CODESYSSPV3/3S/IecVarAccess;String;|var|CODESYS Control Win V3 x64.Application.IOs.SOP720_Pal_Full;Read;SOP720_Pal_Full;Digital;;
CODESYSSPV3/3S/IecVarAccess;String;|var|CODESYS Control Win V3 x64.Application.IOs.SOP720_Pal_Refill;Read;SOP720_Pal_Refill;Digital;;
CODESYSSPV3/3S/IecVarAccess;String;|var|CODESYS Control Win V3 x64.Application.IOs.SOP720_Pal_Dispense;Read;SOP720_Pal_Dispense;Digital;;
CODESYSSPV3/3S/IecVarAccess;String;|var|CODESYS Control Win V3 x64.Application.IOs.SOP721_KM1;Read;SOP721_KM1;Digital;;
CODESYSSPV3/3S/IecVarAccess;String;|var|CODESYS Control Win V3 x64.Application.IOs.SOP721_KM2;Read;SOP721_KM2;Digital;;
CODESYSSPV3/3S/IecVarAccess;String;|var|CODESYS Control Win V3 x64.Application.IOs.SOP730_KM1;Read;SOP730_KM1;Digital;;
CODESYSSPV3/3S/IecVarAccess;String;|var|CODESYS Control Win V3 x64.Application.IOs.SOP730_KM2;Read;SOP730_KM2;Digital;;
CODESYSSPV3/3S/IecVarAccess;String;|var|CODESYS Control Win V3 x64.Application.IOs.SOP730_K2;Read;SOP730_K2;Digital;;
CODESYSSPV3/3S/IecVarAccess;String;|var|CODESYS Control Win V3 x64.Application.IOs.SOP730_K3;Read;SOP730_K3;Digital;;
CODESYSSPV3/3S/IecVarAccess;String;|var|CODESYS Control Win V3 x64.Application.IOs.SOP730_K4;Read;SOP730_K4;Digital;;
CODESYSSPV3/3S/IecVarAccess;String;|var|CODESYS Control Win V3 x64.Application.IOs.SOP730_K5;Read;SOP730_K5;Digital;;
CODESYSSPV3/3S/IecVarAccess;String;|var|CODESYS Control Win V3 x64.Application.IOs.SOP722_KM1;Read;SOP722_KM1;Digital;;
CODESYSSPV3/3S/IecVarAccess;String;|var|CODESYS Control Win V3 x64.Application.IOs.SOP722_KM2;Read;SOP722_KM2;Digital;;
CODESYSSPV3/3S/IecVarAccess;String;|var|CODESYS Control Win V3 x64.Application.IOs.SOP723_KM1;Read;SOP723_KM1;Digital;;
CODESYSSPV3/3S/IecVarAccess;String;|var|CODESYS Control Win V3 x64.Application.IOs.SOP723_KM2;Read;SOP723_KM2;Digital;;
CODESYSSPV3/3S/IecVarAccess;String;|var|CODESYS Control Win V3 x64.Application.IOs.SOP723_K1;Read;SOP723_K1;Digital;;
CODESYSSPV3/3S/IecVarAccess;String;|var|CODESYS Control Win V3 x64.Application.IOs.SOP723_K2;Read;SOP723_K2;Digital;;
CODESYSSPV3/3S/IecVarAccess;String;|var|CODESYS Control Win V3 x64.Application.IOs.SOP740_PickProduct;Read;SOP740_PickProduct;Digital;;
CODESYSSPV3/3S/IecVarAccess;String;|var|CODESYS Control Win V3 x64.Application.IOs.SOP750_K3;Read;SOP750_K3;Digital;;
CODESYSSPV3/3S/IecVarAccess;String;|var|CODESYS Control Win V3 x64.Application.IOs.SOP750_K4;Read;SOP750_K4;Digital;;
CODESYSSPV3/3S/IecVarAccess;String;|var|CODESYS Control Win V3 x64.Application.IOs.SOP750_K5;Read;SOP750_K5;Digital;;
CODESYSSPV3/3S/IecVarAccess;String;|var|CODESYS Control Win V3 x64.Application.IOs.SOP750_K6;Read;SOP750_K6;Digital;;
CODESYSSPV3/3S/IecVarAccess;String;|var|CODESYS Control Win V3 x64.Application.IOs.SOP700_Faulted;Read;SOP700_Faulted;Digital;;
CODESYSSPV3/3S/IecVarAccess;String;|var|CODESYS Control Win V3 x64.Application.IOs.SOP740_Pal_Pos_1;Read;SOP740_Pal_Pos_1;Digital;;
CODESYSSPV3/3S/IecVarAccess;String;|var|CODESYS Control Win V3 x64.Application.IOs.SOP740_Pal_Pos_2;Read;SOP740_Pal_Pos_2;Digital;;
CODESYSSPV3/3S/IecVarAccess;String;|var|CODESYS Control Win V3 x64.Application.IOs.SOP740_Pal_Pos_3;Read;SOP740_Pal_Pos_3;Digital;;
CODESYSSPV3/3S/IecVarAccess;String;|var|CODESYS Control Win V3 x64.Application.IOs.SOP700_H1;Read;SOP700_H1;Digital;;
CODESYSSPV3/3S/IecVarAccess;String;|var|CODESYS Control Win V3 x64.Application.IOs.SOP700_H4;Read;SOP700_H4;Digital;;
CODESYSSPV3/3S/IecVarAccess;String;|var|CODESYS Control Win V3 x64.Application.IOs.SOP700_H7;Read;SOP700_H7;Digital;;
CODESYSSPV3/3S/IecVarAccess;String;|var|CODESYS Control Win V3 x64.Application.IOs.SOP700_H10;Read;SOP700_H10;Digital;;
CODESYSSPV3/3S/IecVarAccess;String;|var|CODESYS Control Win V3 x64.Application.IOs.SOP700_H11;Read;SOP700_H11;Digital;;
CODESYSSPV3/3S/IecVarAccess;String;|var|CODESYS Control Win V3 x64.Application.IOs.SOP700_H14;Read;SOP700_H14;Digital;;
CODESYSSPV3/3S/IecVarAccess;String;|var|CODESYS Control Win V3 x64.Application.IOs.SOP700_H15;Read;SOP700_H15;Digital;;
CODESYSSPV3/3S/IecVarAccess;String;|var|CODESYS Control Win V3 x64.Application.IOs.SOP700_H16;Read;SOP700_H16;Digital;;
CODESYSSPV3/3S/IecVarAccess;String;|var|CODESYS Control Win V3 x64.Application.IOs.SOP740_ProductNr;Read;SOP740_ProductNr;Group;;
CODESYSSPV3/3S/IecVarAccess;String;|var|CODESYS Control Win V3 x64.Application.IOs.SOP723_RetirePallet;Read;SOP723_RetirePallet;Digital;;
CODESYSSPV3/3S/IecVarAccess;String;|var|CODESYS Control Win V3 x64.Application.IOs.SOP720_K5;Read;SOP720_K5;Digital;;
CODESYSSPV3/3S/IecVarAccess;String;|var|CODESYS Control Win V3 x64.Application.IOs.SOP720_K6;Read;SOP720_K6;Digital;;
CODESYSSPV3/3S/IecVarAccess;String;|var|CODESYS Control Win V3 x64.Application.IOs.SOP720_DispensorUp;Write;SOP720_DispensorUp;Digital;;
CODESYSSPV3/3S/IecVarAccess;String;|var|CODESYS Control Win V3 x64.Application.IOs.SOP720_DispensorMid;Write;SOP720_DispensorMid;Digital;;
CODESYSSPV3/3S/IecVarAccess;String;|var|CODESYS Control Win V3 x64.Application.IOs.SOP720_DispensorDown;Write;SOP720_DispensorDown;Digital;;
CODESYSSPV3/3S/IecVarAccess;String;|var|CODESYS Control Win V3 x64.Application.IOs.SOP720_Pal_DispenseDown;Read;SOP720_Pal_DispenseDown;Digital;;
CODESYSSPV3/3S/IecVarAccess;String;|var|CODESYS Control Win V3 x64.Application.IOs.Box_ProductNr;Write;Box_ProductNr;Group;;
CODESYSSPV3/3S/IecVarAccess;String;|var|CODESYS Control Win V3 x64.Application.IOs.Box_IDNumber;Write;Box_IDNumber;Group;;
CODESYSSPV3/3S/IecVarAccess;String;|var|CODESYS Control Win V3 x64.Application.IOs.Status;Write;Status;Group;;

  - Light Curtain Sensor 1 [smart component] at (-31.6, 0, -77.53) mm
      signals: DI DisableSensor, DO Detection
      connections:
        PlaneSensor.SensorOut -> Light Curtain Sensor 1.Detection
        Light Curtain Sensor 1.DisableSensor -> Hide.Execute
        Light Curtain Sensor 1.DisableSensor -> LogicGate_3.InputA
        LogicGate_3.Output -> Show.Execute
        Light Curtain Sensor 1.DisableSensor -> LogicGate_4.InputA
        LogicGate_4.Output -> PlaneSensor.Active
    - PlaneSensor [smart component, from Components\PlaneSensor.rslib] at (2884.52, 14026.71, 333.51) mm, rotated rx 180 ry 0 rz 0 deg
        properties: Origin=[2.28654003266257 4.4307927432671 0.0338898089966275]; Axis1=[2.3 0 0]; Axis2=[0 0 -1.4]; Tag=(none); SensedPart=(none)
      - _sensorPart_ [part], size 2300 x 0 x 1400 mm
    - Show [smart component, from Components\Show.rslib]
        properties: Object=PlaneSensor
    - Hide [smart component, from Components\Hide.rslib]
        properties: Object=PlaneSensor
    - LogicGate_3 [smart component, from Components\LogicGate.rslib]
        properties: Operator=NOT; Delay=0
    - LogicGate_4 [smart component, from Components\LogicGate.rslib]
        properties: Operator=NOT; Delay=0
  - Light Curtain Sensor 2 [smart component] at (0, -1819.31, 0) mm
      signals: DI DisableSensor, DO Detection
      connections:
        PlaneSensor_2.SensorOut -> Light Curtain Sensor 2.Detection
        Light Curtain Sensor 2.DisableSensor -> Show_2.Execute
        Light Curtain Sensor 2.DisableSensor -> LogicGate_4.InputA
        Light Curtain Sensor 2.DisableSensor -> Hide_2.Execute
        LogicGate_4.Output -> Show.Execute
        Light Curtain Sensor 2.DisableSensor -> LogicGate_5.InputA
        LogicGate_5.Output -> PlaneSensor_2.Active
    - PlaneSensor_2 [smart component, from Components\PlaneSensor.rslib] at (0, 0, 396.73) mm
        properties: Origin=[5.139461 9.59591 0.22208]; Axis1=[2.3 0 0]; Axis2=[0 0 1]; Tag=(none); SensedPart=(none)
      - _sensorPart_ [part], size 2300 x 0 x 1000 mm
    - Hide_2 [smart component, from Components\Hide.rslib]
        properties: Object=PlaneSensor_2
    - LogicGate_4 [smart component, from Components\LogicGate.rslib]
        properties: Operator=NOT; Delay=0
    - Show [smart component, from Components\Show.rslib]
        properties: Object=PlaneSensor_2
    - LogicGate_5 [smart component, from Components\LogicGate.rslib]
        properties: Operator=NOT; Delay=0
  - Light Curtain Sensor 3 [smart component] at (0, -6989.64, 0) mm
      signals: DI DisableSensor, DO Detection
      connections:
        PlaneSensor_3.SensorOut -> Light Curtain Sensor 3.Detection
        LogicGate_5.Output -> Show_3.Execute
        Light Curtain Sensor 3.DisableSensor -> Hide_3.Execute
        Light Curtain Sensor 3.DisableSensor -> LogicGate_5.InputA
        LogicGate_5.Output -> PlaneSensor_3.Active
    - PlaneSensor_3 [smart component, from Components\PlaneSensor.rslib] at (-89.72, 0, 389.63) mm
        properties: Origin=[5.139461 9.59591 0.22208]; Axis1=[2.4 0 0]; Axis2=[0 0 1]; Tag=(none); SensedPart=(none)
      - _sensorPart_ [part], size 2400 x 0 x 1000 mm
    - LogicGate_5 [smart component, from Components\LogicGate.rslib]
        properties: Operator=NOT; Delay=0
    - Show_3 [smart component, from Components\Show.rslib]
        properties: Object=PlaneSensor_3
    - Hide_3 [smart component, from Components\Hide.rslib]
        properties: Object=PlaneSensor_3
  - Light Curtain Sensor 4 [smart component] at (17259.69, -4413.54, -135.54) mm, rotated rx 0 ry 0 rz 90 deg
      signals: DI DisableSensor, DO Detection
      connections:
        PlaneSensor_4.SensorOut -> Light Curtain Sensor 4.Detection
        Light Curtain Sensor 4.DisableSensor -> Hide_4.Execute
        Light Curtain Sensor 4.DisableSensor -> LogicGate_6.InputA
        LogicGate_6.Output -> Show_4.Execute
        LogicGate_6.Output -> PlaneSensor_4.Active
    - PlaneSensor_4 [smart component, from Components\PlaneSensor.rslib] at (-119.79, 209.38, 385.64) mm
        properties: Origin=[5.139461 9.59591 0.22208]; Axis1=[2 0 0]; Axis2=[0 0 1.15]; Tag=(none); SensedPart=(none)
      - _sensorPart_ [part], size 2000 x 0 x 1150 mm
    - Hide_4 [smart component, from Components\Hide.rslib]
        properties: Object=PlaneSensor_4
    - Show_4 [smart component, from Components\Show.rslib]
        properties: Object=PlaneSensor_4
    - LogicGate_6 [smart component, from Components\LogicGate.rslib]
        properties: Operator=NOT; Delay=0
  - Timer [smart component, from Components\Timer.rslib]
      properties: StartTime=0; Interval=0; Repeat=true; CurrentTime=6.024
  - MB16 [part] at (-390.31, 2938.54, 153.88) mm, rotated rx -90 ry 0 rz -174.01 deg, size 307.8 x 156.9 x 705.9 mm
  - MB20 [part] at (-193.15, 1001.07, 153.01) mm, rotated rx 0 ry -90 rz 87.74 deg, size 307.4 x 156.7 x 856 mm
  - MB24 [part] at (1.3, -34.41, 112.44) mm, rotated rx 102.56 ry 0 rz -2.8 deg, size 308.5 x 176.3 x 856.1 mm
  - MB16T [part] at (28.49, 2049.11, 116.85) mm, rotated rx 90 ry 0 rz 104.11 deg, size 705.9 x 158.8 x 305.9 mm
  - SOP722 [smart component] at (6333.61, 6970, 616.89) mm, rotated rx 0 ry 0 rz 90 deg
      properties: ForwardSpeed=0.05; ReverseSpeed=-0.05; ConveyorSpeed=0; SpeedForward=0.7; Constant=1E-09; SpeedBackward=-0.6
      signals: DI MotorFWD, DI MotorREV, DO ConveyorError, DI ResetError, DO MotorFeedback, DO BoxSensor
      connections:
        SOP722.MotorFWD -> ?.Enabled
        SOP722.MotorREV -> ?.Enabled
        ?.Output -> ?.Enabled
        SOP722.MotorFWD -> ?.Execute
        SOP722.MotorREV -> ?.Execute
        SOP722.MotorFWD -> ?.A
        SOP722.MotorREV -> ?.B
        ?.Result -> ConveyorSurfaceBehaviour.SurfaceVelocity
        ?.Output -> ConveyorSurfaceBehaviour.SurfaceVelocity
        ?.Output -> ?.InputA
        ?.Output -> ?.InputB
        SOP722.MotorFWD -> ?.InputA
        SOP722.MotorFWD -> ?.InputA
        SOP722.MotorREV -> ?.InputB
        SOP722.MotorFWD -> ?.InputA
        SOP722.MotorFWD -> ?.A
        ?.Result -> ConveyorSurfaceBehaviour.SurfaceVelocity
        SOP722.MotorFWD -> ?.Set
        SOP722.MotorREV -> ?.Set
        SetIdleSpeed.Result -> SetIdleSpeedToConveyor.Execute
        SOP722.MotorFWD -> SetIdleSpeed.A
        SOP722.MotorREV -> SetIdleSpeed.B
        SOP722.MotorFWD -> SetMotorSafetyBreaker.FWD
        SOP722.MotorREV -> SetMotorSafetyBreaker.REV
        ErrorCheckAndBlockingMotorsAndErrorResetLogic.Output -> SetIdleSpeedToConveyor.Execute
        SOP722.ResetError -> ErrorCheckAndBlockingMotorsAndErrorResetLogic.Reset
        SOP722.MotorFWD -> NoErrorAllowFWD.FWD
        ErrorCheckAndBlockingMotorsAndErrorResetLogic.Output -> NoErrorAllowFWD.Error
        NoErrorAllowFWD.Result -> SetForwardSpeedToConveyor.Execute
        SOP722.MotorREV -> NoErrorAllowREV.REV
        ErrorCheckAndBlockingMotorsAndErrorResetLogic.Output -> NoErrorAllowREV.Error
        NoErrorAllowREV.Result -> SetBackwardSpeedToConveyor.Execute
        SetMotorSafetyBreaker.Result -> ErrorCheckAndBlockingMotorsAndErrorResetLogic.Set
        GraphicsHideLogic.Result -> GraphicsHide.Execute
        SOP722.MotorFWD -> GraphicsHideLogic.FWD
        SOP722.MotorREV -> GraphicsHideLogic.REV
        SOP722.MotorFWD -> MotorFeedbackSignalLogic.A
        SOP722.MotorREV -> MotorFeedbackSignalLogic.A
        ErrorCheckAndBlockingMotorsAndErrorResetLogic.Output -> MotorFeedbackSignalLogic.B
        MotorFeedbackSignalLogic.Result -> SOP722.MotorFeedback
        MotorFeedbackSignalLogic.Result -> GraphicsShow.Execute
        ErrorCheckAndBlockingMotorsAndErrorResetLogic.InvOutput -> SOP722.ConveyorError
        SUB100_B1.SensorSignal -> SOP722.BoxSensor
        ?.Result => ?.Count
        ?.Value => ConveyorSurfaceBehaviour.SurfaceVelocity
        ?.Value => ConveyorSurfaceBehaviour.SurfaceVelocity
        ?.Value => ConveyorSurfaceBehaviour.SurfaceVelocity
        ?.Value => ConveyorSurfaceBehaviour.SurfaceVelocity
        ?.Value => ConveyorSurfaceBehaviour.SurfaceVelocity
        ?.Value => ConveyorSurfaceBehaviour.SurfaceVelocity
        SetIdleSpeedToConveyor.Value => ConveyorSurfaceBehaviour.SurfaceVelocity
        SetForwardSpeedToConveyor.Value => ConveyorSurfaceBehaviour.SurfaceVelocity
        SetBackwardSpeedToConveyor.Value => ConveyorSurfaceBehaviour.SurfaceVelocity
        ?.Result => SetForwardSpeedToConveyor.Max
        ?.A => SetBackwardSpeedToConveyor.Min
        ?.Result => SetBackwardSpeedToConveyor.Max
        ?.A => SetForwardSpeedToConveyor.Min
        GraphicsShow.Object => GraphicsHide.Object
        ?.Object => ?.Object
    - ConveyorSurfaceBehaviour [smart component, from Components\PhysicsControl.rslib] at (-850.96, -505.17, -100) mm
        properties: Object=ConveyorSurface; Behavior=2; SurfaceVelocity=0.500000000078149
    - SetIdleSpeedToConveyor [smart component, from Components\Random.rslib] at (-850.96, -505.17, -100) mm
        properties: Value=3.63538950385311E-14; Min=0; Max=1E-13
    - SetBackwardSpeedToConveyor [smart component, from Components\Random.rslib] at (-850.96, -505.17, -100) mm
        properties: Value=-0.699999999999963; Min=-0.7; Max=-0.6999999999999
    - SetForwardSpeedToConveyor [smart component, from Components\Random.rslib] at (-850.96, -505.17, -100) mm
        properties: Value=0.500000000078149; Min=0.5; Max=0.5000000001
    - SetIdleSpeed [smart component, from Components\LogicExpression.rslib] at (-850.96, -505.17, -100) mm
        properties: Expression=not A and not B
    - SetMotorSafetyBreaker [smart component, from Components\LogicExpression.rslib] at (-850.96, -505.17, -100) mm
        properties: Expression=FWD and REV
    - ErrorCheckAndBlockingMotorsAndErrorResetLogic [smart component, from Components\LogicSRLatch.rslib] at (-850.96, -505.17, -100) mm
    - NoErrorAllowFWD [smart component, from Components\LogicExpression.rslib] at (-850.96, -505.17, -100) mm
        properties: Expression=FWD and not Error
    - NoErrorAllowREV [smart component, from Components\LogicExpression.rslib] at (-850.96, -505.17, -100) mm
        properties: Expression=REV and not Error
    - GraphicsShow [smart component, from Components\Show.rslib] at (-850.96, -505.17, -100) mm
        properties: Object=OnOffGfx
    - GraphicsHide [smart component, from Components\Hide.rslib] at (-850.96, -505.17, -100) mm
        properties: Object=OnOffGfx
    - GraphicsHideLogic [smart component, from Components\LogicExpression.rslib] at (-850.96, -505.17, -100) mm
        properties: Expression=not FWD and not REV
    - GraphicsObjects [graphiccomponentgroup] at (-65.23, -0.94, 0) mm, rotated rx 0 ry 0 rz -90 deg
      - OnOffGfx [graphiccomponentgroup] at (514.42, -850.96, -110.92) mm, rotated rx 0 ry 0 rz 90 deg
        - Part_5 [part] at (-19.01, -85.34, -416.89) mm, rotated rx 0 ry 0 rz -90 deg, size 50 x 1701.5 x 100 mm
        - Part_6 [part] at (0, 1062.79, 0) mm, rotated rx 0 ry 0 rz -90 deg, size 50 x 1701.5 x 100 mm
      - ConveyorSurface [part] at (505.17, -850.96, -112.36) mm, rotated rx 0 ry 0 rz 90 deg, size 1712.3 x 1089.6 x 114.1 mm
    - MotorFeedbackSignalLogic [smart component, from Components\LogicExpression.rslib] at (-850.96, -505.17, -100) mm
        properties: Expression=A AND NOT B
    - Conveyor [part] at (-916.73, -600.7, -162.63) mm, rotated rx 0 ry 0 rz 180 deg, size 1700 x 1300 x 500 mm
    - SUB100_B1 [smart component] at (565.82, 599.25, -101.36) mm, rotated rx 0 ry 0 rz 180 deg
        signals: DO SensorSignal
        connections:
          SensorRay.SensorOut -> ?.Active
          ?.Output -> SUB100_B1.SensorSignal
          SensorRay.SensorOut -> LogicGate.InputA
          GraphicSwitch_2.Output -> LogicGate_2.InputA
          LogicGate_2.Output -> LogicGate.InputB
          LogicGate.Output -> SUB100_B1.SensorSignal
      - SensorRay [smart component, from Components\LineSensor.rslib] at (24.04, 61.94, 174.13) mm
          properties: Start=[0 0 0]; End=[5.26116255894493E-07 0.938058416436489 2.90984203399347E-08]; Radius=0.01; SensedPart=(none); SensedPoint=[0 0 0]; Length=0.938058416436637; Tag=(none)
        - _sensorPart_ [part], size 20 x 938.1 x 20 mm
      - SensorMountWorking [part] at (0, 0, 0) mm, size 50 x 50 x 200 mm
      - GraphicSwitch_2 [smart component, from Components\GraphicSwitch.rslib] at (50, 0, 0) mm
          properties: PartHigh=SensorMountBroken; PartLow=SensorMountWorking
      - SensorMountBroken [part] at (0, 0, 0) mm, size 50 x 50 x 200 mm
      - LogicGate [smart component, from Components\LogicGate.rslib]
          properties: Operator=AND; Delay=0
      - LogicGate_2 [smart component, from Components\LogicGate.rslib]
          properties: Operator=NOT; Delay=0
  - SOP723 [smart component] at (6335.13, 8670, 616.89) mm, rotated rx 0 ry 0 rz 90 deg
      properties: ForwardSpeed=0.05; ReverseSpeed=-0.05; ConveyorSpeed=0; SpeedForward=0.7; Constant=1E-09; SpeedBackward=-0.6
      signals: DI MotorFWD, DI MotorREV, DO ConveyorError, DI ResetError, DO MotorFeedback, DO BoxSensor
      connections:
        SOP723.MotorFWD -> ?.Enabled
        SOP723.MotorREV -> ?.Enabled
        ?.Output -> ?.Enabled
        SOP723.MotorFWD -> ?.Execute
        SOP723.MotorREV -> ?.Execute
        SOP723.MotorFWD -> ?.A
        SOP723.MotorREV -> ?.B
        ?.Result -> ConveyorSurfaceBehaviour.SurfaceVelocity
        ?.Output -> ConveyorSurfaceBehaviour.SurfaceVelocity
        ?.Output -> ?.InputA
        ?.Output -> ?.InputB
        SOP723.MotorFWD -> ?.InputA
        SOP723.MotorFWD -> ?.InputA
        SOP723.MotorREV -> ?.InputB
        SOP723.MotorFWD -> ?.InputA
        SOP723.MotorFWD -> ?.A
        ?.Result -> ConveyorSurfaceBehaviour.SurfaceVelocity
        SOP723.MotorFWD -> ?.Set
        SOP723.MotorREV -> ?.Set
        SetIdleSpeed.Result -> SetIdleSpeedToConveyor.Execute
        SOP723.MotorFWD -> SetIdleSpeed.A
        SOP723.MotorREV -> SetIdleSpeed.B
        SOP723.MotorFWD -> SetMotorSafetyBreaker.FWD
        SOP723.MotorREV -> SetMotorSafetyBreaker.REV
        ErrorCheckAndBlockingMotorsAndErrorResetLogic.Output -> SetIdleSpeedToConveyor.Execute
        SOP723.ResetError -> ErrorCheckAndBlockingMotorsAndErrorResetLogic.Reset
        SOP723.MotorFWD -> NoErrorAllowFWD.FWD
        ErrorCheckAndBlockingMotorsAndErrorResetLogic.Output -> NoErrorAllowFWD.Error
        NoErrorAllowFWD.Result -> SetForwardSpeedToConveyor.Execute
        SOP723.MotorREV -> NoErrorAllowREV.REV
        ErrorCheckAndBlockingMotorsAndErrorResetLogic.Output -> NoErrorAllowREV.Error
        NoErrorAllowREV.Result -> SetBackwardSpeedToConveyor.Execute
        SetMotorSafetyBreaker.Result -> ErrorCheckAndBlockingMotorsAndErrorResetLogic.Set
        GraphicsHideLogic.Result -> GraphicsHide.Execute
        SOP723.MotorFWD -> GraphicsHideLogic.FWD
        SOP723.MotorREV -> GraphicsHideLogic.REV
        SOP723.MotorFWD -> MotorFeedbackSignalLogic.A
        SOP723.MotorREV -> MotorFeedbackSignalLogic.A
        ErrorCheckAndBlockingMotorsAndErrorResetLogic.Output -> MotorFeedbackSignalLogic.B
        MotorFeedbackSignalLogic.Result -> SOP723.MotorFeedback
        MotorFeedbackSignalLogic.Result -> GraphicsShow.Execute
        ErrorCheckAndBlockingMotorsAndErrorResetLogic.InvOutput -> SOP723.ConveyorError
        SUB100_B1.SensorSignal -> SOP723.BoxSensor
        ?.Result => ?.Count
        ?.Value => ConveyorSurfaceBehaviour.SurfaceVelocity
        ?.Value => ConveyorSurfaceBehaviour.SurfaceVelocity
        ?.Value => ConveyorSurfaceBehaviour.SurfaceVelocity
        ?.Value => ConveyorSurfaceBehaviour.SurfaceVelocity
        ?.Value => ConveyorSurfaceBehaviour.SurfaceVelocity
        ?.Value => ConveyorSurfaceBehaviour.SurfaceVelocity
        SetIdleSpeedToConveyor.Value => ConveyorSurfaceBehaviour.SurfaceVelocity
        SetForwardSpeedToConveyor.Value => ConveyorSurfaceBehaviour.SurfaceVelocity
        SetBackwardSpeedToConveyor.Value => ConveyorSurfaceBehaviour.SurfaceVelocity
        ?.Result => SetForwardSpeedToConveyor.Max
        ?.A => SetBackwardSpeedToConveyor.Min
        ?.Result => SetBackwardSpeedToConveyor.Max
        ?.A => SetForwardSpeedToConveyor.Min
        GraphicsShow.Object => GraphicsHide.Object
        ?.Object => ?.Object
    - ConveyorSurfaceBehaviour [smart component, from Components\PhysicsControl.rslib] at (-850.96, -505.17, -100) mm
        properties: Object=ConveyorSurface; Behavior=2; SurfaceVelocity=0.500000000006195
    - SetIdleSpeedToConveyor [smart component, from Components\Random.rslib] at (-850.96, -505.17, -100) mm
        properties: Value=1.83222603138174E-14; Min=0; Max=1E-13
    - SetBackwardSpeedToConveyor [smart component, from Components\Random.rslib] at (-850.96, -505.17, -100) mm
        properties: Value=-0.699999999999983; Min=-0.7; Max=-0.6999999999999
    - SetForwardSpeedToConveyor [smart component, from Components\Random.rslib] at (-850.96, -505.17, -100) mm
        properties: Value=0.500000000006195; Min=0.5; Max=0.5000000001
    - SetIdleSpeed [smart component, from Components\LogicExpression.rslib] at (-850.96, -505.17, -100) mm
        properties: Expression=not A and not B
    - SetMotorSafetyBreaker [smart component, from Components\LogicExpression.rslib] at (-850.96, -505.17, -100) mm
        properties: Expression=FWD and REV
    - ErrorCheckAndBlockingMotorsAndErrorResetLogic [smart component, from Components\LogicSRLatch.rslib] at (-850.96, -505.17, -100) mm
    - NoErrorAllowFWD [smart component, from Components\LogicExpression.rslib] at (-850.96, -505.17, -100) mm
        properties: Expression=FWD and not Error
    - NoErrorAllowREV [smart component, from Components\LogicExpression.rslib] at (-850.96, -505.17, -100) mm
        properties: Expression=REV and not Error
    - GraphicsShow [smart component, from Components\Show.rslib] at (-850.96, -505.17, -100) mm
        properties: Object=OnOffGfx
    - GraphicsHide [smart component, from Components\Hide.rslib] at (-850.96, -505.17, -100) mm
        properties: Object=OnOffGfx
    - GraphicsHideLogic [smart component, from Components\LogicExpression.rslib] at (-850.96, -505.17, -100) mm
        properties: Expression=not FWD and not REV
    - GraphicsObjects [graphiccomponentgroup] at (-65.23, -0.94, 0) mm, rotated rx 0 ry 0 rz -90 deg
      - OnOffGfx [graphiccomponentgroup] at (514.42, -850.96, -110.92) mm, rotated rx 0 ry 0 rz 90 deg
        - Part_5 [part] at (-19.01, -85.34, -416.89) mm, rotated rx 0 ry 0 rz -90 deg, size 50 x 1701.5 x 100 mm
        - Part_6 [part] at (0, 1062.79, 0) mm, rotated rx 0 ry 0 rz -90 deg, size 50 x 1701.5 x 100 mm
      - ConveyorSurface [part] at (505.17, -850.96, -112.36) mm, rotated rx 0 ry 0 rz 90 deg, size 1712.3 x 1089.6 x 114.1 mm
    - MotorFeedbackSignalLogic [smart component, from Components\LogicExpression.rslib] at (-850.96, -505.17, -100) mm
        properties: Expression=A AND NOT B
    - Conveyor [part] at (-916.73, -600.7, -162.63) mm, rotated rx 0 ry 0 rz 180 deg, size 1700 x 1300 x 500 mm
    - SUB100_B1 [smart component] at (565.82, 599.25, -101.36) mm, rotated rx 0 ry 0 rz 180 deg
        signals: DO SensorSignal
        connections:
          SensorRay.SensorOut -> ?.Active
          ?.Output -> SUB100_B1.SensorSignal
          SensorRay.SensorOut -> LogicGate.InputA
          GraphicSwitch_2.Output -> LogicGate_2.InputA
          LogicGate_2.Output -> LogicGate.InputB
          LogicGate.Output -> SUB100_B1.SensorSignal
      - SensorRay [smart component, from Components\LineSensor.rslib] at (24.04, 61.94, 174.13) mm
          properties: Start=[0 0 0]; End=[5.26116255894493E-07 0.938058416436489 2.90984203399347E-08]; Radius=0.01; SensedPart=(none); SensedPoint=[0 0 0]; Length=0.938058416436637; Tag=(none)
        - _sensorPart_ [part], size 20 x 938.1 x 20 mm
      - SensorMountWorking [part] at (0, 0, 0) mm, size 50 x 50 x 200 mm
      - GraphicSwitch_2 [smart component, from Components\GraphicSwitch.rslib] at (50, 0, 0) mm
          properties: PartHigh=SensorMountBroken; PartLow=SensorMountWorking
      - SensorMountBroken [part] at (0, 0, 0) mm, size 50 x 50 x 200 mm
      - LogicGate [smart component, from Components\LogicGate.rslib]
          properties: Operator=AND; Delay=0
      - LogicGate_2 [smart component, from Components\LogicGate.rslib]
          properties: Operator=NOT; Delay=0
  - PalletDispensorMovement [smart component]
      signals: DI ReFillPallet, DI Pallet_FilledUp, DI NewPallet, DO DispensorDown, DO DispensorMid, DO DispensorUp, DI Dispensor_Down, DO DispensorTop
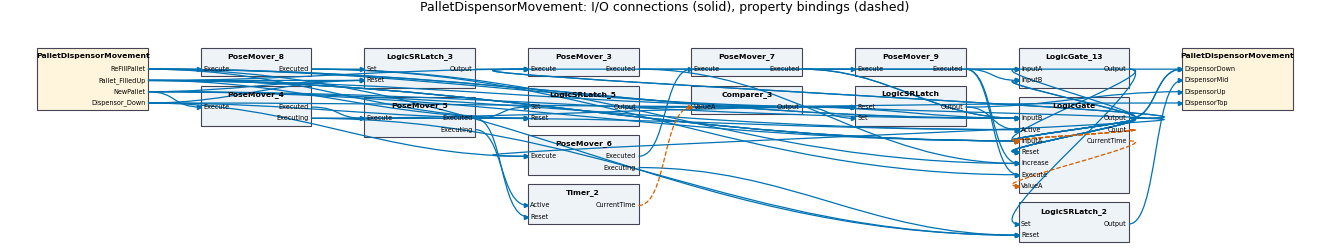
      connections:
        PoseMover_4.Executed -> PoseMover_5.Execute
        PoseMover_6.Executed -> PoseMover_7.Execute
        LogicGate.Output -> PoseMover_3.Execute
        PoseMover_7.Executed -> LogicGate.InputB
        PoseMover_7.Executed -> LogicGate_2.InputB
        LogicGate_2.Output -> PoseMover_3.Execute
        PoseMover_5.Executed -> Timer.Active
        Timer.Output -> PoseMover_6.Execute
        Timer_2.Output -> LogicGate.InputA
        LogicGate.Output -> Timer.Reset
        PalletDispensorMovement.ReFillPallet -> PoseMover_8.Execute
        PalletDispensorMovement.Pallet_FilledUp -> ?.InputA
        PalletDispensorMovement.Pallet_FilledUp -> ?.InputA
        PalletDispensorMovement.Pallet_FilledUp -> PoseMover_3.Execute
        PalletDispensorMovement.NewPallet -> PoseMover_4.Execute
        PalletDispensorMovement.NewPallet -> Timer_2.Active
        PoseMover_7.Executed -> PoseMover_9.Execute
        PoseMover_8.Executed -> Counter_2.Increase
        LogicGate_7.Output -> LogicGate_8.InputA
        LogicGate_8.Output -> Counter_2.Reset
        LogicGate_7.Output -> PalletDispensorMovement.DispensorDown
        PoseMover_9.Executed -> Counter_4.Increase
        LogicGate_11.Output -> LogicGate_12.InputA
        LogicGate_12.Output -> Counter_4.Reset
        PoseMover_3.Executed -> Counter_3.Increase
        LogicGate_9.Output -> LogicGate_10.InputA
        LogicGate_10.Output -> Counter_3.Reset
        LogicGate_9.Output -> LogicGate_13.InputA
        LogicGate_11.Output -> LogicGate_13.InputB
        PoseMover_5.Executing -> Timer_2.Active
        PoseMover_5.Executed -> Timer_2.Reset
        PoseMover_9.Executed -> Repeater.Execute
        Repeater.Output -> LogicGate_13.InputB
        PoseMover_8.Executed -> Repeater_2.Execute
        Repeater_2.Output -> PalletDispensorMovement.DispensorDown
        LogicSRLatch.Output -> Timer_4.Active
        Comparer_4.Output -> LogicSRLatch.Reset
        Comparer_4.Output -> Timer_4.Reset
        LogicSRLatch_3.Output -> PalletDispensorMovement.DispensorDown
        LogicSRLatch_2.Output -> PalletDispensorMovement.DispensorMid
        LogicSRLatch.Output -> PalletDispensorMovement.DispensorUp
        Comparer_3.Output -> LogicSRLatch.Set
        PoseMover_8.Executed -> LogicSRLatch_3.Set
        PoseMover_3.Executed -> LogicGate_13.InputA
        PoseMover_9.Executed -> LogicGate_13.InputB
        LogicGate_13.Output -> LogicSRLatch_2.Set
        LogicGate_13.Output -> LogicGate_15.InputA
        PalletDispensorMovement.ReFillPallet -> LogicGate_15.InputB
        PalletDispensorMovement.Pallet_FilledUp -> LogicGate_14.InputA
        PalletDispensorMovement.NewPallet -> LogicGate_14.InputB
        PalletDispensorMovement.NewPallet -> LogicGate_16.InputA
        PalletDispensorMovement.ReFillPallet -> LogicGate_16.InputB
        LogicGate_16.Output -> LogicGate_17.InputA
        Comparer_3.Output -> LogicGate_17.InputB
        PalletDispensorMovement.Dispensor_Down -> PoseMover_6.Execute
        PoseMover_5.Executed -> LogicSRLatch_5.Set
        LogicSRLatch_5.Output -> PalletDispensorMovement.DispensorTop
        PalletDispensorMovement.ReFillPallet -> LogicSRLatch.Reset
        PalletDispensorMovement.Pallet_FilledUp -> LogicSRLatch.Reset
        PalletDispensorMovement.Dispensor_Down -> LogicSRLatch.Reset
        PoseMover_4.Executing -> LogicSRLatch.Reset
        PalletDispensorMovement.ReFillPallet -> LogicSRLatch_5.Reset
        PalletDispensorMovement.Pallet_FilledUp -> LogicSRLatch_5.Reset
        PalletDispensorMovement.Dispensor_Down -> LogicSRLatch_5.Reset
        PoseMover_4.Executing -> LogicSRLatch_5.Reset
        PalletDispensorMovement.ReFillPallet -> LogicSRLatch_2.Reset
        PoseMover_4.Executing -> LogicSRLatch_2.Reset
        PoseMover_6.Executing -> LogicSRLatch_2.Reset
        PalletDispensorMovement.Pallet_FilledUp -> LogicSRLatch_3.Reset
        PalletDispensorMovement.NewPallet -> LogicSRLatch_3.Reset
        PalletDispensorMovement.Dispensor_Down -> LogicSRLatch_3.Reset
        LogicSRLatch_5.Output -> LogicSRLatch.Reset
        Counter_2.Count => LogicGate_7.InputA
        Counter_4.Count => LogicGate_11.InputA
        Counter_3.Count => LogicGate_9.InputA
        Timer_2.CurrentTime => Comparer_3.ValueA
        Timer_4.CurrentTime => Comparer_4.ValueA
    - PoseMover_3 [smart component, from Components\PoseMover.rslib]
        properties: Mechanism=PalletDispenser; Pose=2; Duration=2
    - PoseMover_4 [smart component, from Components\PoseMover.rslib]
        properties: Mechanism=PalletDispenser; Pose=3; Duration=2
    - PoseMover_5 [smart component, from Components\PoseMover.rslib]
        properties: Mechanism=PalletDispenser; Pose=4; Duration=4
    - PoseMover_6 [smart component, from Components\PoseMover.rslib]
        properties: Mechanism=PalletDispenser; Pose=5; Duration=4
    - PoseMover_7 [smart component, from Components\PoseMover.rslib]
        properties: Mechanism=PalletDispenser; Pose=6; Duration=2
    - PoseMover_8 [smart component, from Components\PoseMover.rslib]
        properties: Mechanism=PalletDispenser; Pose=1; Duration=1
    - PoseMover_9 [smart component, from Components\PoseMover.rslib]
        properties: Mechanism=PalletDispenser; Pose=2; Duration=2
    - LogicGate_13 [smart component, from Components\LogicGate.rslib]
        properties: Operator=OR; Delay=0
    - Timer_2 [smart component, from Components\Timer.rslib]
        properties: StartTime=0; Interval=0; Repeat=true; CurrentTime=0
    - Comparer_3 [smart component, from Components\Comparer.rslib]
        properties: ValueA=0; Operator=>=; ValueB=1
    - LogicSRLatch [smart component, from Components\LogicSRLatch.rslib]
    - LogicSRLatch_2 [smart component, from Components\LogicSRLatch.rslib]
    - LogicSRLatch_3 [smart component, from Components\LogicSRLatch.rslib]
    - LogicSRLatch_5 [smart component, from Components\LogicSRLatch.rslib]
  - PalletDispenser [mechanism] at (0, 0, 0) mm; joint values [0.1316, 0, 0] (rad or m)
      links: Wall, HorizontalBar, LeftClamp, RightClamp
  - EuroPallet (1) [part] at (8313.49, 1114.92, 117.23) mm, rotated rx 0 ry 0 rz 89.94 deg, size 1206.6 x 808.8 x 152.5 mm
  - Buttons [graphiccomponentgroup]
    - FilledPallet [part] at (7471.38, 607.83, 1076.55) mm, rotated rx 0 ry 90 rz 0 deg, size 40 x 39.8 x 10 mm
    - Emergency4 [part] at (7471.38, 607.83, 1236.44) mm, rotated rx 0 ry 90 rz 0 deg, size 40 x 39.8 x 10 mm
    - PalletRemove [part] at (7441.66, 9631.65, 1174.65) mm, rotated rx 0 ry 90 rz 90 deg, size 40 x 39.8 x 10 mm
    - Emergency3 [part] at (7441.66, 9631.65, 1280.76) mm, rotated rx 0 ry 90 rz 90 deg, size 40 x 39.8 x 10 mm
    - Emergency1 [part] at (5192.96, 10430.05, 1449.33) mm, rotated rx 0 ry 90 rz -180 deg, size 40 x 39.8 x 10 mm
    - Emergency2 [part] at (5138.96, 10431.72, 1432.3) mm, rotated rx 0 ry 90 rz -180 deg, size 40 x 39.8 x 10 mm
  - SOP730 [smart component] at (6335.96, 5270, 616.89) mm, rotated rx 0 ry 0 rz 90 deg
      properties: ForwardSpeed=0.05; ReverseSpeed=-0.05; ConveyorSpeed=0; SpeedForward=0.7; Constant=1E-09; SpeedBackward=-0.6
      signals: DI MotorFWD, DI MotorREV, DO ConveyorError, DI ResetError, DO MotorFeedback, DI FrontUp, DI FrontDown, DI RearUp, DI RearDown, DO BoxSensor, DO FrontSensor, DO RearSensor, DO FrontDownSensor, DO RareDownSensor
      connections:
        SOP730.MotorFWD -> ?.Enabled
        SOP730.MotorREV -> ?.Enabled
        ?.Output -> ?.Enabled
        SOP730.MotorFWD -> ?.Execute
        SOP730.MotorREV -> ?.Execute
        SOP730.MotorFWD -> ?.A
        SOP730.MotorREV -> ?.B
        ?.Result -> ConveyorSurfaceBehaviour.SurfaceVelocity
        ?.Output -> ConveyorSurfaceBehaviour.SurfaceVelocity
        ?.Output -> ?.InputA
        ?.Output -> ?.InputB
        SOP730.MotorFWD -> ?.InputA
        SOP730.MotorFWD -> ?.InputA
        SOP730.MotorREV -> ?.InputB
        SOP730.MotorFWD -> ?.InputA
        SOP730.MotorFWD -> ?.A
        ?.Result -> ConveyorSurfaceBehaviour.SurfaceVelocity
        SOP730.MotorFWD -> ?.Set
        SOP730.MotorREV -> ?.Set
        SetIdleSpeed.Result -> SetIdleSpeedToConveyor.Execute
        SOP730.MotorFWD -> SetIdleSpeed.A
        SOP730.MotorREV -> SetIdleSpeed.B
        SOP730.MotorFWD -> SetMotorSafetyBreaker.FWD
        SOP730.MotorREV -> SetMotorSafetyBreaker.REV
        ErrorCheckAndBlockingMotorsAndErrorResetLogic.Output -> SetIdleSpeedToConveyor.Execute
        SOP730.ResetError -> ErrorCheckAndBlockingMotorsAndErrorResetLogic.Reset
        SOP730.MotorFWD -> NoErrorAllowFWD.FWD
        ErrorCheckAndBlockingMotorsAndErrorResetLogic.Output -> NoErrorAllowFWD.Error
        NoErrorAllowFWD.Result -> SetForwardSpeedToConveyor.Execute
        SOP730.MotorREV -> NoErrorAllowREV.REV
        ErrorCheckAndBlockingMotorsAndErrorResetLogic.Output -> NoErrorAllowREV.Error
        NoErrorAllowREV.Result -> SetBackwardSpeedToConveyor.Execute
        SetMotorSafetyBreaker.Result -> ErrorCheckAndBlockingMotorsAndErrorResetLogic.Set
        GraphicsHideLogic.Result -> GraphicsHide.Execute
        SOP730.MotorFWD -> GraphicsHideLogic.FWD
        SOP730.MotorREV -> GraphicsHideLogic.REV
        SOP730.MotorFWD -> MotorFeedbackSignalLogic.A
        SOP730.MotorREV -> MotorFeedbackSignalLogic.A
        ErrorCheckAndBlockingMotorsAndErrorResetLogic.Output -> MotorFeedbackSignalLogic.B
        MotorFeedbackSignalLogic.Result -> SOP730.MotorFeedback
        MotorFeedbackSignalLogic.Result -> GraphicsShow.Execute
        ErrorCheckAndBlockingMotorsAndErrorResetLogic.InvOutput -> SOP730.ConveyorError
        SUB100_B1.SensorSignal -> SOP730.BoxSensor
        SUB730 FrontClamp.ClampUpPosition -> SOP730.FrontSensor
        SUB730 RearClamp.ClampUpPosition -> SOP730.RearSensor
        SOP730.FrontUp -> SUB730 FrontClamp.ClampUp
        SOP730.FrontDown -> SUB730 FrontClamp.ClampDown
        SOP730.RearUp -> SUB730 RearClamp.ClampUp
        SOP730.RearDown -> SUB730 RearClamp.ClampDown
        SOP730.FrontUp -> SUB730 FrontClamp.ClampUp
        SOP730.FrontDown -> SUB730 FrontClamp.ClampDown
        SUB730 FrontClamp.ClampUpPosition -> SOP730.FrontSensor
        SOP730.RearUp -> SUB730 RearClamp.ClampUp
        SOP730.RearDown -> SUB730 RearClamp.ClampDown
        SUB730 RearClamp.ClampUpPosition -> SOP730.RearSensor
        SUB730 FrontClamp.ClampDownPosition -> SOP730.FrontDownSensor
        SUB730 RearClamp.ClampDownPosition -> SOP730.RareDownSensor
        SOP730.FrontUp -> SUB730 FrontClamp.ClampUp
        SOP730.FrontDown -> SUB730 FrontClamp.ClampDown
        SUB730 FrontClamp.ClampUpPosition -> SOP730.FrontSensor
        SUB730 FrontClamp.ClampDownPosition -> SOP730.FrontDownSensor
        ?.Result => ?.Count
        ?.Value => ConveyorSurfaceBehaviour.SurfaceVelocity
        ?.Value => ConveyorSurfaceBehaviour.SurfaceVelocity
        ?.Value => ConveyorSurfaceBehaviour.SurfaceVelocity
        ?.Value => ConveyorSurfaceBehaviour.SurfaceVelocity
        ?.Value => ConveyorSurfaceBehaviour.SurfaceVelocity
        ?.Value => ConveyorSurfaceBehaviour.SurfaceVelocity
        SetIdleSpeedToConveyor.Value => ConveyorSurfaceBehaviour.SurfaceVelocity
        SetForwardSpeedToConveyor.Value => ConveyorSurfaceBehaviour.SurfaceVelocity
        SetBackwardSpeedToConveyor.Value => ConveyorSurfaceBehaviour.SurfaceVelocity
        ?.Result => SetForwardSpeedToConveyor.Max
        ?.A => SetBackwardSpeedToConveyor.Min
        ?.Result => SetBackwardSpeedToConveyor.Max
        ?.A => SetForwardSpeedToConveyor.Min
        GraphicsShow.Object => GraphicsHide.Object
        ?.Object => ?.Object
    - ConveyorSurfaceBehaviour [smart component, from Components\PhysicsControl.rslib] at (-850.96, -505.17, -100) mm
        properties: Object=ConveyorSurface; Behavior=2; SurfaceVelocity=0.500000000050282
    - SetIdleSpeedToConveyor [smart component, from Components\Random.rslib] at (-850.96, -505.17, -100) mm
        properties: Value=6.11436496307811E-14; Min=0; Max=1E-13
    - SetBackwardSpeedToConveyor [smart component, from Components\Random.rslib] at (-850.96, -505.17, -100) mm
        properties: Value=-0.699999999999912; Min=-0.7; Max=-0.6999999999999
    - SetForwardSpeedToConveyor [smart component, from Components\Random.rslib] at (-850.96, -505.17, -100) mm
        properties: Value=0.500000000050282; Min=0.5; Max=0.5000000001
    - SetIdleSpeed [smart component, from Components\LogicExpression.rslib] at (-850.96, -505.17, -100) mm
        properties: Expression=not A and not B
    - SetMotorSafetyBreaker [smart component, from Components\LogicExpression.rslib] at (-850.96, -505.17, -100) mm
        properties: Expression=FWD and REV
    - ErrorCheckAndBlockingMotorsAndErrorResetLogic [smart component, from Components\LogicSRLatch.rslib] at (-850.96, -505.17, -100) mm
    - NoErrorAllowFWD [smart component, from Components\LogicExpression.rslib] at (-850.96, -505.17, -100) mm
        properties: Expression=FWD and not Error
    - NoErrorAllowREV [smart component, from Components\LogicExpression.rslib] at (-850.96, -505.17, -100) mm
        properties: Expression=REV and not Error
    - GraphicsShow [smart component, from Components\Show.rslib] at (-850.96, -505.17, -100) mm
        properties: Object=OnOffGfx
    - GraphicsHide [smart component, from Components\Hide.rslib] at (-850.96, -505.17, -100) mm
        properties: Object=OnOffGfx
    - GraphicsHideLogic [smart component, from Components\LogicExpression.rslib] at (-850.96, -505.17, -100) mm
        properties: Expression=not FWD and not REV
    - GraphicsObjects [graphiccomponentgroup] at (-65.23, -0.94, 0) mm, rotated rx 0 ry 0 rz -90 deg
      - OnOffGfx [graphiccomponentgroup] at (514.42, -850.96, -110.92) mm, rotated rx 0 ry 0 rz 90 deg
        - Part_5 [part] at (-19.01, -85.34, -416.89) mm, rotated rx 0 ry 0 rz -90 deg, size 50 x 1701.5 x 100 mm
        - Part_6 [part] at (0, 1062.79, 0) mm, rotated rx 0 ry 0 rz -90 deg, size 50 x 1701.5 x 100 mm
      - ConveyorSurface [part] at (505.17, -850.96, -112.36) mm, rotated rx 0 ry 0 rz 90 deg, size 1712.3 x 1089.6 x 114.1 mm
    - MotorFeedbackSignalLogic [smart component, from Components\LogicExpression.rslib] at (-850.96, -505.17, -100) mm
        properties: Expression=A AND NOT B
    - Conveyor [part] at (-916.73, -600.7, -162.63) mm, rotated rx 0 ry 0 rz 180 deg, size 1700 x 1300 x 500 mm
    - SUB100_B1 [smart component] at (565.82, 599.25, -101.36) mm, rotated rx 0 ry 0 rz 180 deg
        signals: DO SensorSignal
        connections:
          SensorRay.SensorOut -> ?.Active
          ?.Output -> SUB100_B1.SensorSignal
          SensorRay.SensorOut -> LogicGate.InputA
          GraphicSwitch_2.Output -> LogicGate_2.InputA
          LogicGate_2.Output -> LogicGate.InputB
          LogicGate.Output -> SUB100_B1.SensorSignal
      - SensorRay [smart component, from Components\LineSensor.rslib] at (24.04, 61.94, 174.13) mm
          properties: Start=[0 0 0]; End=[5.26116255894493E-07 0.938058416436489 2.90984203399347E-08]; Radius=0.01; SensedPart=(none); SensedPoint=[0 0 0]; Length=0.938058416436637; Tag=(none)
        - _sensorPart_ [part], size 20 x 938.1 x 20 mm
      - SensorMountWorking [part] at (0, 0, 0) mm, size 50 x 50 x 200 mm
      - GraphicSwitch_2 [smart component, from Components\GraphicSwitch.rslib] at (50, 0, 0) mm
          properties: PartHigh=SensorMountBroken; PartLow=SensorMountWorking
      - SensorMountBroken [part] at (0, 0, 0) mm, size 50 x 50 x 200 mm
      - LogicGate [smart component, from Components\LogicGate.rslib]
          properties: Operator=AND; Delay=0
      - LogicGate_2 [smart component, from Components\LogicGate.rslib]
          properties: Operator=NOT; Delay=0
    - SUB730 RearClamp [smart component, from Components\SUB730 RearClamp1.rslib] at (-679.81, -100.54, -122.63) mm, rotated rx 0 ry 0 rz 90 deg
        connections:
          SUB730 RearClamp.ClampUp -> LogicExpression.A
          BottomPosSensor.SensorOut -> LogicExpression.B
          LogicExpression.Result -> LinearMoveUp.Execute
          SUB730 RearClamp.ClampDown -> LogicExpression_2.A
          BottomPosSensor.SensorOut -> LogicExpression_2.B
          LogicExpression_2.Result -> LinearMoveDown.Execute
          LinearMoveUp.Executed -> LogicSRLatch.Set
          LogicSRLatch.Output -> SUB730 RearClamp.ClampUpPosition
          LinearMoveDown.Executed -> ?.Set
          ?.Output -> SUB730 RearClamp.ClampDownPosition
          LinearMoveDown.Executing -> LogicSRLatch.Reset
          LinearMoveUp.Executing -> ?.Reset
          BottomPosSensor.SensorOut -> SUB730 RearClamp.ClampDownPosition
      - Clamp3D [part, from Components\SUB730 RearClamp1.rslib]
      - BottomPosSensor [smart component, from Components\LineSensor.rslib] at (18.37, 10.91, 93.4) mm
          properties: Start=[-5.44677247749092E-09 -9.84894448774476E-08 -0.0999997155196143]; End=[-5.44677247749092E-09 -9.84894448774476E-08 -0.0899997155196144]; Radius=0.02; SensedPart=Clamp3D; SensedPoint=[6.41812744140625 4.57928466796875 0.49426123046875]; Length=0.0099999999999999; Tag=(none)
        - _sensorPart_ [part, from Components\SUB730 RearClamp1.rslib]
      - LinearMoveUp [smart component, from Components\LinearMover2.rslib]
          properties: Object=Clamp3D; Direction=[0 0 0.1]; Distance=0.1; Duration=1; Reference=Global; ReferenceObject=(none)
      - LinearMoveDown [smart component, from Components\LinearMover2.rslib]
          properties: Object=Clamp3D; Direction=[0 0 -0.1]; Distance=0.1; Duration=1; Reference=Global; ReferenceObject=(none)
      - LogicExpression [smart component, from Components\LogicExpression.rslib]
          properties: Expression=A AND B
      - LogicExpression_2 [smart component, from Components\LogicExpression.rslib]
          properties: Expression=A AND NOT B
      - LogicSRLatch [smart component, from Components\LogicSRLatch.rslib]
    - SUB730 FrontClamp [smart component, from Components\SUB730 RearClamp1.rslib] at (571.35, -100.54, -122.63) mm, rotated rx 0 ry 0 rz 90 deg
        connections:
          SUB730 FrontClamp.ClampUp -> LogicExpression.A
          BottomPosSensor.SensorOut -> LogicExpression.B
          LogicExpression.Result -> LinearMoveUp.Execute
          SUB730 FrontClamp.ClampDown -> LogicExpression_2.A
          BottomPosSensor.SensorOut -> LogicExpression_2.B
          LogicExpression_2.Result -> LinearMoveDown.Execute
          LinearMoveUp.Executed -> LogicSRLatch.Set
          LogicSRLatch.Output -> SUB730 FrontClamp.ClampUpPosition
          LinearMoveDown.Executed -> ?.Set
          ?.Output -> SUB730 FrontClamp.ClampDownPosition
          LinearMoveDown.Executing -> LogicSRLatch.Reset
          LinearMoveUp.Executing -> ?.Reset
          BottomPosSensor.SensorOut -> SUB730 FrontClamp.ClampDownPosition
      - Clamp3D [part, from Components\SUB730 RearClamp1.rslib]
      - BottomPosSensor [smart component, from Components\LineSensor.rslib] at (18.37, 10.91, 93.4) mm
          properties: Start=[-5.44677247749092E-09 -9.84894448774476E-08 -0.0999997155196143]; End=[-5.44677247749092E-09 -9.84894448774476E-08 -0.0899997155196144]; Radius=0.02; SensedPart=Clamp3D; SensedPoint=[6.41812744140625 5.83044482421875 0.494260986328125]; Length=0.0099999999999999; Tag=(none)
        - _sensorPart_ [part, from Components\SUB730 RearClamp1.rslib]
      - LinearMoveUp [smart component, from Components\LinearMover2.rslib]
          properties: Object=Clamp3D; Direction=[0 0 0.1]; Distance=0.1; Duration=1; Reference=Global; ReferenceObject=(none)
      - LinearMoveDown [smart component, from Components\LinearMover2.rslib]
          properties: Object=Clamp3D; Direction=[0 0 -0.1]; Distance=0.1; Duration=1; Reference=Global; ReferenceObject=(none)
      - LogicExpression [smart component, from Components\LogicExpression.rslib]
          properties: Expression=A AND B
      - LogicExpression_2 [smart component, from Components\LogicExpression.rslib]
          properties: Expression=A AND NOT B
      - LogicSRLatch [smart component, from Components\LogicSRLatch.rslib]
  - SOP721 [smart component] at (6333.61, 3570, 616.89) mm, rotated rx 0 ry 0 rz 90 deg
      properties: ForwardSpeed=0.05; ReverseSpeed=-0.05; ConveyorSpeed=0; SpeedForward=0.7; Constant=1E-09; SpeedBackward=-0.6
      signals: DI MotorFWD, DI MotorREV, DO ConveyorError, DI ResetError, DO MotorFeedback, DO BoxSensor
      connections:
        SOP721.MotorFWD -> ?.Enabled
        SOP721.MotorREV -> ?.Enabled
        ?.Output -> ?.Enabled
        SOP721.MotorFWD -> ?.Execute
        SOP721.MotorREV -> ?.Execute
        SOP721.MotorFWD -> ?.A
        SOP721.MotorREV -> ?.B
        ?.Result -> ConveyorSurfaceBehaviour.SurfaceVelocity
        ?.Output -> ConveyorSurfaceBehaviour.SurfaceVelocity
        ?.Output -> ?.InputA
        ?.Output -> ?.InputB
        SOP721.MotorFWD -> ?.InputA
        SOP721.MotorFWD -> ?.InputA
        SOP721.MotorREV -> ?.InputB
        SOP721.MotorFWD -> ?.InputA
        SOP721.MotorFWD -> ?.A
        ?.Result -> ConveyorSurfaceBehaviour.SurfaceVelocity
        SOP721.MotorFWD -> ?.Set
        SOP721.MotorREV -> ?.Set
        SetIdleSpeed.Result -> SetIdleSpeedToConveyor.Execute
        SOP721.MotorFWD -> SetIdleSpeed.A
        SOP721.MotorREV -> SetIdleSpeed.B
        SOP721.MotorFWD -> SetMotorSafetyBreaker.FWD
        SOP721.MotorREV -> SetMotorSafetyBreaker.REV
        ErrorCheckAndBlockingMotorsAndErrorResetLogic.Output -> SetIdleSpeedToConveyor.Execute
        SOP721.ResetError -> ErrorCheckAndBlockingMotorsAndErrorResetLogic.Reset
        SOP721.MotorFWD -> NoErrorAllowFWD.FWD
        ErrorCheckAndBlockingMotorsAndErrorResetLogic.Output -> NoErrorAllowFWD.Error
        NoErrorAllowFWD.Result -> SetForwardSpeedToConveyor.Execute
        SOP721.MotorREV -> NoErrorAllowREV.REV
        ErrorCheckAndBlockingMotorsAndErrorResetLogic.Output -> NoErrorAllowREV.Error
        NoErrorAllowREV.Result -> SetBackwardSpeedToConveyor.Execute
        SetMotorSafetyBreaker.Result -> ErrorCheckAndBlockingMotorsAndErrorResetLogic.Set
        GraphicsHideLogic.Result -> GraphicsHide.Execute
        SOP721.MotorFWD -> GraphicsHideLogic.FWD
        SOP721.MotorREV -> GraphicsHideLogic.REV
        SOP721.MotorFWD -> MotorFeedbackSignalLogic.A
        SOP721.MotorREV -> MotorFeedbackSignalLogic.A
        ErrorCheckAndBlockingMotorsAndErrorResetLogic.Output -> MotorFeedbackSignalLogic.B
        MotorFeedbackSignalLogic.Result -> SOP721.MotorFeedback
        MotorFeedbackSignalLogic.Result -> GraphicsShow.Execute
        ErrorCheckAndBlockingMotorsAndErrorResetLogic.InvOutput -> SOP721.ConveyorError
        SUB100_B1.SensorSignal -> SOP721.BoxSensor
        ?.Result => ?.Count
        ?.Value => ConveyorSurfaceBehaviour.SurfaceVelocity
        ?.Value => ConveyorSurfaceBehaviour.SurfaceVelocity
        ?.Value => ConveyorSurfaceBehaviour.SurfaceVelocity
        ?.Value => ConveyorSurfaceBehaviour.SurfaceVelocity
        ?.Value => ConveyorSurfaceBehaviour.SurfaceVelocity
        ?.Value => ConveyorSurfaceBehaviour.SurfaceVelocity
        SetIdleSpeedToConveyor.Value => ConveyorSurfaceBehaviour.SurfaceVelocity
        SetForwardSpeedToConveyor.Value => ConveyorSurfaceBehaviour.SurfaceVelocity
        SetBackwardSpeedToConveyor.Value => ConveyorSurfaceBehaviour.SurfaceVelocity
        ?.Result => SetForwardSpeedToConveyor.Max
        ?.A => SetBackwardSpeedToConveyor.Min
        ?.Result => SetBackwardSpeedToConveyor.Max
        ?.A => SetForwardSpeedToConveyor.Min
        GraphicsShow.Object => GraphicsHide.Object
        ?.Object => ?.Object
    - ConveyorSurfaceBehaviour [smart component, from Components\PhysicsControl.rslib] at (-850.96, -505.17, -100) mm
        properties: Object=ConveyorSurface; Behavior=2; SurfaceVelocity=0.500000000015493
    - SetIdleSpeedToConveyor [smart component, from Components\Random.rslib] at (-850.96, -505.17, -100) mm
        properties: Value=0; Min=0; Max=1E-13
    - SetBackwardSpeedToConveyor [smart component, from Components\Random.rslib] at (-850.96, -505.17, -100) mm
        properties: Value=-0.699999999999991; Min=-0.7; Max=-0.6999999999999
    - SetForwardSpeedToConveyor [smart component, from Components\Random.rslib] at (-850.96, -505.17, -100) mm
        properties: Value=0.500000000015493; Min=0.5; Max=0.5000000001
    - SetIdleSpeed [smart component, from Components\LogicExpression.rslib] at (-850.96, -505.17, -100) mm
        properties: Expression=not A and not B
    - SetMotorSafetyBreaker [smart component, from Components\LogicExpression.rslib] at (-850.96, -505.17, -100) mm
        properties: Expression=FWD and REV
    - ErrorCheckAndBlockingMotorsAndErrorResetLogic [smart component, from Components\LogicSRLatch.rslib] at (-850.96, -505.17, -100) mm
    - NoErrorAllowFWD [smart component, from Components\LogicExpression.rslib] at (-850.96, -505.17, -100) mm
        properties: Expression=FWD and not Error
    - NoErrorAllowREV [smart component, from Components\LogicExpression.rslib] at (-850.96, -505.17, -100) mm
        properties: Expression=REV and not Error
    - GraphicsShow [smart component, from Components\Show.rslib] at (-850.96, -505.17, -100) mm
        properties: Object=OnOffGfx
    - GraphicsHide [smart component, from Components\Hide.rslib] at (-850.96, -505.17, -100) mm
        properties: Object=OnOffGfx
    - GraphicsHideLogic [smart component, from Components\LogicExpression.rslib] at (-850.96, -505.17, -100) mm
        properties: Expression=not FWD and not REV
    - GraphicsObjects [graphiccomponentgroup] at (-65.23, -0.94, 0) mm, rotated rx 0 ry 0 rz -90 deg
      - OnOffGfx [graphiccomponentgroup] at (514.42, -850.96, -110.92) mm, rotated rx 0 ry 0 rz 90 deg
        - Part_5 [part] at (-19.01, -85.34, -416.89) mm, rotated rx 0 ry 0 rz -90 deg, size 50 x 1701.5 x 100 mm
        - Part_6 [part] at (0, 1062.79, 0) mm, rotated rx 0 ry 0 rz -90 deg, size 50 x 1701.5 x 100 mm
      - ConveyorSurface [part] at (505.17, -850.96, -112.36) mm, rotated rx 0 ry 0 rz 90 deg, size 1712.3 x 1089.6 x 114.1 mm
    - MotorFeedbackSignalLogic [smart component, from Components\LogicExpression.rslib] at (-850.96, -505.17, -100) mm
        properties: Expression=A AND NOT B
    - Conveyor [part] at (-916.73, -600.7, -162.63) mm, rotated rx 0 ry 0 rz 180 deg, size 1700 x 1300 x 500 mm
    - SUB100_B1 [smart component, from Components\SUB100_B1.rslib] at (565.82, 599.25, -101.36) mm, rotated rx 0 ry 0 rz 180 deg
        connections:
          SensorRay.SensorOut -> ?.Active
          ?.Output -> SUB100_B1.SensorSignal
          SensorRay.SensorOut -> LogicGate.InputA
          GraphicSwitch_2.Output -> LogicGate_2.InputA
          LogicGate_2.Output -> LogicGate.InputB
          LogicGate.Output -> SUB100_B1.SensorSignal
      - SensorRay [smart component, from Components\LineSensor.rslib] at (24.04, 61.94, 174.13) mm
          properties: Start=[0 0 0]; End=[5.26116255894493E-07 0.938058416436489 2.90984203399347E-08]; Radius=0.01; SensedPart=(none); SensedPoint=[0 0 0]; Length=0.938058416436637; Tag=(none)
        - _sensorPart_ [part, from Components\SUB100_B1.rslib]
      - SensorMountWorking [part, from Components\SUB100_B1.rslib] at (0, 0, 0) mm
      - GraphicSwitch_2 [smart component, from Components\GraphicSwitch.rslib] at (50, 0, 0) mm
          properties: PartHigh=SensorMountBroken; PartLow=SensorMountWorking
      - SensorMountBroken [part, from Components\SUB100_B1.rslib] at (0, 0, 0) mm
      - LogicGate [smart component, from Components\LogicGate.rslib]
          properties: Operator=AND; Delay=0
      - LogicGate_2 [smart component, from Components\LogicGate.rslib]
          properties: Operator=NOT; Delay=0
  - IRB4400_60_196__03 [mechanism] at (4963.29, 5843.46, 0) mm, rotated rx 0 ry 0 rz -90 deg; joint values [0, 0, 0, 0, 0.5236, 0] (rad or m)
      links: Base, Link1, Link2, Link3, Link4, Link5, Link6, LinkD1, LinkD2, LinkD3, LinkD4
  - sensor_730front [smart component, from Components\LineSensor.rslib]
      properties: Start=[6.244 5.975 0.665]; End=[6.444 5.975 0.665]; Length=0.2; Radius=0; Tag=(none); SensedPart=(none); SensedPoint=[0 0 0]
    - _sensorPart_ [part], size 200 x 0 x 0 mm
  - sensor_730rare [smart component, from Components\LineSensor.rslib]
      properties: Start=[6.244 4.58 0.66]; End=[6.444 4.58 0.66]; Length=0.2; Radius=0; Tag=(none); SensedPart=(none); SensedPoint=[0 0 0]
    - _sensorPart_ [part], size 200 x 0 x 0 mm
  - sensor_713front [smart component, from Components\LineSensor.rslib]
      properties: Start=[3.94 5.796 1.158]; End=[4.14 5.796 1.158]; Length=0.2; Radius=0; Tag=(none); SensedPart=Clamp3D; SensedPoint=[4.12034912109375 5.796 1.158]
    - _sensorPart_ [part], size 200 x 0 x 0 mm
  - sensor_713rare [smart component, from Components\LineSensor.rslib]
      properties: Start=[3.92 4.795 1.158]; End=[4.12 4.795 1.158]; Length=0.2; Radius=0; Tag=(none); SensedPart=Clamp3D; SensedPoint=[3.92034912109375 4.795 1.158]
    - _sensorPart_ [part], size 200 x 0 x 0 mm
  - vacuum [mechanism] at (4963.29, 4642.22, 1650) mm, rotated rx 180 ry 60 rz 90 deg
      TCP vacuum at (0, 0, 175) mm
      links: PalletizingVacuumTool
  - OP710 Input Product [smart component]
      signals: GO ProductNr, GO IDNumber, GO Status, DO AckProductInPlace, DI ResetProductData, DI Create_MB16T, DI Create_MB20, DI Create_MB24, DI Create_MB16, DI sensor717, DI sensor723, DI VacuumOn_I, DI Reject_MB16, DI Reject_MB16T, DI Reject_MB20, DI Reject_MB24, DI RetirePallet
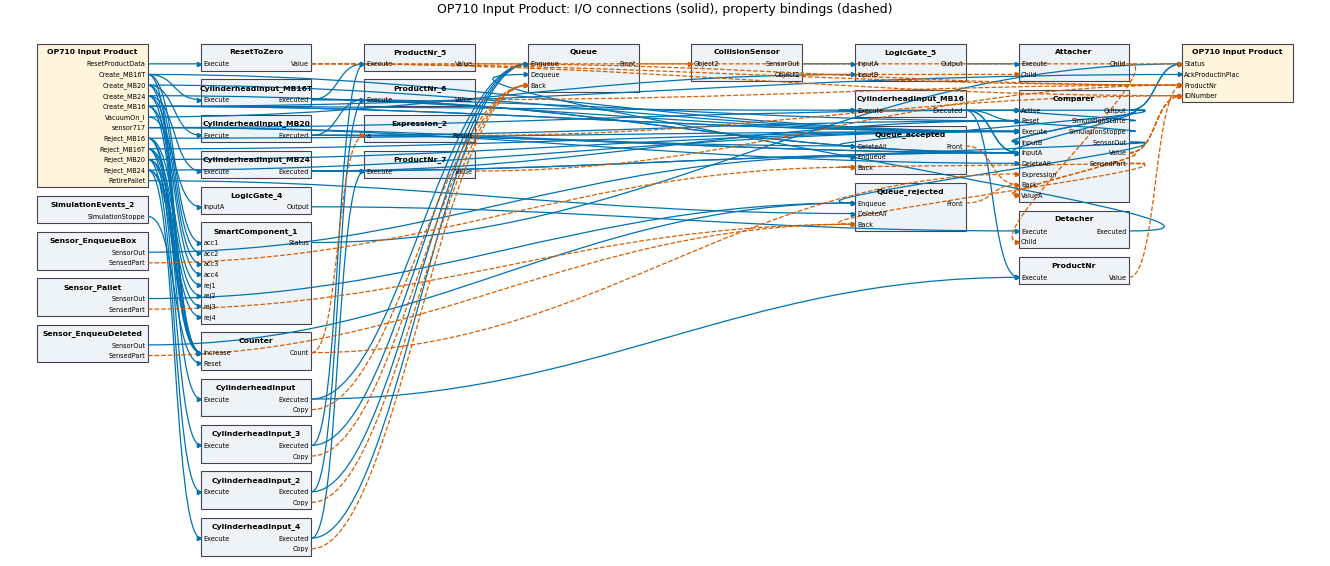
      connections:
        OP710 Input Product.ResetProductData -> ResetToZero.Execute
        Comparer.Output -> OP710 Input Product.Status
        CylinderheadInput_MB16.Executed -> ProductNr.Execute
        CylinderheadInput_MB16T.Executed -> ProductNr_5.Execute
        CylinderheadInput_MB24.Executed -> ProductNr_7.Execute
        CylinderheadInput_MB20.Executed -> ProductNr_6.Execute
        SimulationEvents.SimulationStarted -> Timer.Active
        Timer.Output -> CylinderheadInput_MB16.Execute
        SimulationEvents.SimulationStopped -> Timer.Reset
        OP710 Input Product.Create_MB16T -> CylinderheadInput_MB16T.Execute
        OP710 Input Product.Create_MB20 -> CylinderheadInput_MB20.Execute
        OP710 Input Product.Create_MB24 -> CylinderheadInput_MB24.Execute
        OP710 Input Product.Create_MB16 -> CylinderheadInput_MB16.Execute
        OP710 Input Product.Create_MB16 -> IDNumber.Execute
        OP710 Input Product.Create_MB16 -> OP710 Input Product.AckProductInPlace
        OP710 Input Product.Create_MB16T -> Counter.Increase
        OP710 Input Product.Create_MB20 -> Counter.Increase
        OP710 Input Product.Create_MB24 -> Counter.Increase
        OP710 Input Product.Create_MB16 -> Counter.Increase
        SimulationEvents_2.SimulationStopped -> Counter.Reset
        Comparer.Output -> LogicGate.InputB
        Comparer.Output -> LogicGate_3.InputA
        LogicGate_3.Output -> LogicGate_2.InputB
        CylinderheadInput_MB16T.Executed -> LogicGate.InputA
        CylinderheadInput_MB24.Executed -> LogicGate.InputA
        CylinderheadInput_MB24.Executed -> LogicGate_2.InputA
        CylinderheadInput_MB16T.Executed -> LogicGate_2.InputA
        CylinderheadInput_MB16.Executed -> LogicGate.InputA
        CylinderheadInput_MB20.Executed -> LogicGate.InputA
        CylinderheadInput_MB16.Executed -> LogicGate_2.InputA
        CylinderheadInput_MB20.Executed -> LogicGate_2.InputA
        OP710 Input Product.VacuumOn_I -> LogicGate_4.InputA
        LogicGate_4.Output -> Detacher.Execute
        LogicGate_5.Output -> Attacher.Execute
        CollisionSensor.SensorOut -> LogicGate_5.InputA
        OP710 Input Product.VacuumOn_I -> LogicGate_5.InputB
        Timer_3.Output -> Queue_accepted.DeleteAll
        OP710 Input Product.sensor717 -> Timer_3.Active
        CylinderheadInput_MB16.Executed -> Timer_3.Reset
        CylinderheadInput_MB16T.Executed -> Timer_3.Reset
        CylinderheadInput_MB20.Executed -> Timer_3.Reset
        CylinderheadInput_MB24.Executed -> Timer_3.Reset
        OP710 Input Product.Create_MB16T -> Status.Execute
        OP710 Input Product.Create_MB24 -> Status.Execute
        OP710 Input Product.Create_MB20 -> Status.Execute
        OP710 Input Product.Create_MB16 -> Status.Execute
        OP710 Input Product.sensor717 -> Queue.DeleteAll
        Comparer_2.Output -> OP710 Input Product.Status
        CylinderheadInput.Executed -> ProductNr.Execute
        OP710 Input Product.Reject_MB16 -> CylinderheadInput.Execute
        OP710 Input Product.Reject_MB16 -> Status_2.Execute
        OP710 Input Product.Reject_MB16T -> Status_2.Execute
        OP710 Input Product.Reject_MB20 -> Status_2.Execute
        OP710 Input Product.Reject_MB24 -> Status_2.Execute
        CylinderheadInput_2.Executed -> ProductNr_6.Execute
        OP710 Input Product.Reject_MB20 -> CylinderheadInput_2.Execute
        CylinderheadInput_3.Executed -> ProductNr_5.Execute
        OP710 Input Product.Reject_MB16T -> CylinderheadInput_3.Execute
        OP710 Input Product.Reject_MB16 -> Counter.Increase
        OP710 Input Product.Reject_MB16T -> Counter.Increase
        OP710 Input Product.Reject_MB20 -> Counter.Increase
        OP710 Input Product.Reject_MB24 -> Counter.Increase
        CylinderheadInput_4.Executed -> ProductNr_7.Execute
        OP710 Input Product.Reject_MB24 -> CylinderheadInput_4.Execute
        LineSensor_11.SensorOut -> Queue_accepted.Enqueue
        Sensor_EnqueueRejected.SensorOut -> Queue_rejected.Enqueue
        Sensor_EnqueueBox.SensorOut -> Queue_accepted.Enqueue
        OP710 Input Product.Create_MB16T -> SmartComponent_1.acc1
        OP710 Input Product.Create_MB20 -> SmartComponent_1.acc2
        OP710 Input Product.Create_MB24 -> SmartComponent_1.acc3
        OP710 Input Product.Create_MB16 -> SmartComponent_1.acc4
        OP710 Input Product.Reject_MB16 -> SmartComponent_1.rej1
        OP710 Input Product.Reject_MB16T -> SmartComponent_1.rej2
        OP710 Input Product.Reject_MB20 -> SmartComponent_1.rej3
        OP710 Input Product.Reject_MB24 -> SmartComponent_1.rej4
        OP710 Input Product.sensor717 -> Queue_accepted.DeleteAll
        CylinderheadInput.Executed -> Queue.Enqueue
        CylinderheadInput_2.Executed -> Queue.Enqueue
        CylinderheadInput_3.Executed -> Queue.Enqueue
        CylinderheadInput_4.Executed -> Queue.Enqueue
        Detacher.Executed -> Queue.Dequeue
        Sensor_Pallet.SensorOut -> Queue_rejected.Enqueue
        Sensor_EnqueuDeleted.SensorOut -> Queue_rejected.Enqueue
        OP710 Input Product.RetirePallet -> Queue_rejected.DeleteAll
        SmartComponent_1.Status -> OP710 Input Product.Status
        ProductNr.Value => OP710 Input Product.ProductNr
        ResetToZero.Value => OP710 Input Product.ProductNr
        ResetToZero.Value => OP710 Input Product.IDNumber
        ResetToZero.Value => OP710 Input Product.Status
        ProductNr_5.Value => OP710 Input Product.ProductNr
        IDNumber_5.Value => OP710 Input Product.IDNumber
        ProductNr_6.Value => OP710 Input Product.ProductNr
        IDNumber_6.Value => OP710 Input Product.IDNumber
        ProductNr_7.Value => OP710 Input Product.ProductNr
        IDNumber_7.Value => OP710 Input Product.IDNumber
        Counter.Count => Expression_2.Expression
        Queue_accepted.Front => Queue.Back
        Queue_rejected.Front => Queue_2.Back
        Status.Value => Comparer.ValueA
        Status_2.Value => Comparer_2.ValueA
        LineSensor_11.SensedPart => Queue_accepted.Back
        Sensor_EnqueueRejected.SensedPart => Queue_rejected.Back
        Sensor_EnqueueBox.SensedPart => Queue_accepted.Back
        Counter.Count => Expression_2.a
        Expression_2.Result => OP710 Input Product.IDNumber
        CollisionSensor.Object2 => Attacher.Child
        Attacher.Child => Detacher.Child
        CylinderheadInput.Copy => Queue.Back
        CylinderheadInput_2.Copy => Queue.Back
        CylinderheadInput_4.Copy => Queue.Back
        Queue.Front => CollisionSensor.Object2
        CylinderheadInput_3.Copy => Queue.Back
        Sensor_EnqueuDeleted.SensedPart => Queue_rejected.Back
        Sensor_Pallet.SensedPart => Queue_rejected.Back
    - CylinderheadInput_MB16 [smart component, from Components\Source.rslib]
        properties: Source=MB16; Copy=(none); Parent=(none); Position=[4.025 1.018 1.086]; Orientation=[1.5707963267949 0 0]; Transient=false; PhysicsBehavior=3
    - MB24 [part, from Components\MB24.rslib] at (0, -1189.46, 0) mm
    - ProductNr [smart component, from Components\Random.rslib]
        properties: Value=1604.99850009723; Min=1604.99; Max=1605
    - ResetToZero [smart component, from Components\Random.rslib]
        properties: Value=7.62012279947294E-11; Min=0; Max=1E-09
    - CylinderheadInput_MB16T [smart component, from Components\Source.rslib]
        properties: Source=MB16T; Copy=(none); Parent=(none); Position=[4.025 1.018 1.086]; Orientation=[1.5707963267949 0 1.5707963267949]; Transient=false; PhysicsBehavior=3
    - CylinderheadInput_MB20 [smart component, from Components\Source.rslib]
        properties: Source=MB20; Copy=(none); Parent=(none); Position=[4.025 1.018 1.086]; Orientation=[1.5707963267949 0 0]; Transient=false; PhysicsBehavior=3
    - CylinderheadInput_MB24 [smart component, from Components\Source.rslib]
        properties: Source=MB24; Copy=(none); Parent=(none); Position=[4.025 1.018 1.086]; Orientation=[1.5707963267949 0 0]; Transient=false; PhysicsBehavior=3
    - ProductNr_5 [smart component, from Components\Random.rslib]
        properties: Value=1609.99351505082; Min=1609.99; Max=1610
    - ProductNr_6 [smart component, from Components\Random.rslib]
        properties: Value=2003.99144637039; Min=2003.99; Max=2004
    - ProductNr_7 [smart component, from Components\Random.rslib]
        properties: Value=2406.99999915089; Min=2406.999999; Max=2407
    - Counter [smart component, from Components\Counter.rslib]
        properties: Count=0
    - SimulationEvents_2 [smart component, from Components\SimulationEvents.rslib]
    - Queue_rejected [smart component, from Components\Queue.rslib]
        properties: Back=(none); Front=(none); Queue={ececd2ae-751b-45d0-b5da-bc69544dd414}; NumberOfObjects=1
    - Queue_accepted [smart component, from Components\Queue.rslib]
        properties: Back=(none); Front=(none); Queue=; NumberOfObjects=0
    - Detacher [smart component, from Components\Detacher.rslib]
        properties: Child=(none); KeepPosition=true
    - Attacher [smart component, from Components\Attacher.rslib]
        properties: Parent=vacuum; Flange=0; Child=(none); Mount=false; Offset=[0 0 0]; Orientation=[0 0 0]
    - LogicGate_4 [smart component, from Components\LogicGate.rslib]
        properties: Operator=NOT; Delay=0
    - CollisionSensor [smart component, from Components\CollisionSensor.rslib]
        properties: Object1=vacuum; Object2=(none); NearMiss=0.001; Part1=PalletizingVacuumTool; Part2=Link6; CollisionType=2
    - LogicGate_5 [smart component, from Components\LogicGate.rslib]
        properties: Operator=AND; Delay=0
    - CylinderheadInput [smart component, from Components\Source.rslib]
        properties: Source=MB16; Copy=(none); Parent=(none); Position=[4.025 1.018 1.086]; Orientation=[1.5707963267949 0 0]; Transient=false; PhysicsBehavior=3
    - CylinderheadInput_2 [smart component, from Components\Source.rslib]
        properties: Source=MB20; Copy=(none); Parent=(none); Position=[4.025 1.018 1.086]; Orientation=[1.5707963267949 0 0]; Transient=false; PhysicsBehavior=3
    - CylinderheadInput_3 [smart component, from Components\Source.rslib]
        properties: Source=MB16T; Copy=(none); Parent=(none); Position=[4.025 1.018 1.086]; Orientation=[1.5707963267949 0 1.5707963267949]; Transient=false; PhysicsBehavior=3
    - CylinderheadInput_4 [smart component, from Components\Source.rslib]
        properties: Source=MB24; Copy=(none); Parent=(none); Position=[4.025 1.018 1.086]; Orientation=[1.5707963267949 0 0]; Transient=false; PhysicsBehavior=3
    - Sensor_EnqueueBox [smart component, from Components\PlaneSensor.rslib]
        properties: Origin=[3.92 10.3 1.14]; Axis1=[0.1 0 0]; Axis2=[0 0.1 0]; Tag=(none); SensedPart=(none)
      - _sensorPart_ [part], size 100 x 100 x 0 mm
    - SmartComponent_1 [smart component]
        signals: DI acc1, DI acc2, DI acc3, DI acc4, DI rej1, DI rej2, DI rej3, DI rej4, GO Status
        connections:
          SmartComponent_1.acc1 -> LogicGate.InputA
          SmartComponent_1.acc2 -> LogicGate.InputB
          SmartComponent_1.acc3 -> LogicGate_2.InputA
          SmartComponent_1.acc4 -> LogicGate_2.InputB
          LogicGate.Output -> LogicGate_3.InputA
          LogicGate_2.Output -> LogicGate_3.InputB
          LogicGate_4.Output -> LogicGate_6.InputA
          LogicGate_5.Output -> LogicGate_6.InputB
          SmartComponent_1.rej1 -> LogicGate_4.InputA
          SmartComponent_1.rej2 -> LogicGate_4.InputB
          SmartComponent_1.rej3 -> LogicGate_5.InputA
          SmartComponent_1.rej4 -> LogicGate_5.InputB
          LogicGate_6.Output -> Counter.Increase
          LogicGate_3.Output -> Counter.Reset
          LogicGate_3.Output -> LogicSRLatch.Set
          LogicSRLatch.Output -> Expression.a
          SmartComponent_1.rej1 -> LogicGate_4.InputA
          SmartComponent_1.rej2 -> LogicGate_4.InputB
          SmartComponent_1.rej3 -> LogicGate_5.InputA
          SmartComponent_1.rej4 -> LogicGate_5.InputB
          LogicGate_4.Output -> LogicGate_6.InputA
          LogicGate_5.Output -> LogicGate_6.InputB
          LogicGate_6.Output -> LogicSRLatch.Reset
          Counter.Count => Comparer.ValueA
          Counter.Count => SmartComponent_1.status
          Expression.Result => SmartComponent_1.status
          Expression.Result => SmartComponent_1.Status
      - LogicGate [smart component, from Components\LogicGate.rslib]
          properties: Operator=OR; Delay=0
      - LogicGate_2 [smart component, from Components\LogicGate.rslib]
          properties: Operator=OR; Delay=0
      - LogicGate_3 [smart component, from Components\LogicGate.rslib]
          properties: Operator=OR; Delay=0
      - Expression [smart component, from Components\Expression.rslib]
          properties: Expression=a*64; Result=0; a=0
      - LogicSRLatch [smart component, from Components\LogicSRLatch.rslib]
      - LogicGate_4 [smart component, from Components\LogicGate.rslib]
          properties: Operator=OR; Delay=0
      - LogicGate_5 [smart component, from Components\LogicGate.rslib]
          properties: Operator=OR; Delay=0
      - LogicGate_6 [smart component, from Components\LogicGate.rslib]
          properties: Operator=OR; Delay=0
    - Sensor_Delete717 [smart component, from Components\PlaneSensor.rslib]
        properties: Origin=[3.92 11.85 1.14]; Axis1=[0 0.1 0]; Axis2=[0.1 0 0]; Tag=(none); SensedPart=(none)
      - _sensorPart_ [part], size 100 x 100 x 0 mm
    - Expression_2 [smart component, from Components\Expression.rslib]
        properties: Expression=100125000+a; Result=100125000; a=0
    - Queue [smart component, from Components\Queue.rslib]
        properties: Back=(none); Front=(none); Queue={8ea377cd-0867-4de7-848c-ece66973d8d0};{63d4bcad-becc-4287-abe8-969ff060f041};{48720447-2da2-45b5-87cc-dac214d89a38};{0044870d-68d7-4f8d-bbcb-29d440aad4b9};{b56791cc-fe53-4844-8ea1-4c8344f2b3a4};{3f832083-e9c9-4b92-8dfb-6875a914d572}; NumberOfObjects=1
    - Queue_4 [smart component, from Components\Queue.rslib]
        properties: Back=(none); Front=(none); Queue=; NumberOfObjects=0
    - Sensor_EnqueuDeleted [smart component, from Components\PlaneSensor.rslib]
        properties: Origin=[6.14626 7.921323 0.832016]; Axis1=[0 0 0.05]; Axis2=[0.4 0 0]; Tag=(none); SensedPart=(none)
      - _sensorPart_ [part], size 400 x 0 x 50 mm
    - Sensor_Pallet [smart component, from Components\PlaneSensor.rslib]
        properties: Origin=[6.14626 7.921323 0.642016]; Axis1=[0 0 0.05]; Axis2=[0.4 0 0]; Tag=(none); SensedPart=(none)
      - _sensorPart_ [part], size 400 x 0 x 50 mm
  - SOP717 [smart component] at (3750, 11820, 100) mm, rotated rx 0 ry 0 rz 90 deg
      properties: ForwardSpeed=0.05; ReverseSpeed=-0.05; ConveyorSpeed=0; SpeedForward=0.7; Constant=1E-09; SpeedBackward=-0.6
      signals: DI MotorFWD, DI MotorREV, DO ConveyorError, DI ResetError, DO MotorFeedback, DO BoxSensor
      connections:
        SOP717.MotorFWD -> ?.Enabled
        SOP717.MotorREV -> ?.Enabled
        ?.Output -> ?.Enabled
        SOP717.MotorFWD -> ?.Execute
        SOP717.MotorREV -> ?.Execute
        SOP717.MotorFWD -> ?.A
        SOP717.MotorREV -> ?.B
        ?.Result -> ConveyorSurfaceBehaviour.SurfaceVelocity
        ?.Output -> ConveyorSurfaceBehaviour.SurfaceVelocity
        ?.Output -> ?.InputA
        ?.Output -> ?.InputB
        SOP717.MotorFWD -> ?.InputA
        SOP717.MotorFWD -> ?.InputA
        SOP717.MotorREV -> ?.InputB
        SOP717.MotorFWD -> ?.InputA
        SOP717.MotorFWD -> ?.A
        ?.Result -> ConveyorSurfaceBehaviour.SurfaceVelocity
        SOP717.MotorFWD -> ?.Set
        SOP717.MotorREV -> ?.Set
        SetIdleSpeed.Result -> SetIdleSpeedToConveyor.Execute
        SOP717.MotorFWD -> SetIdleSpeed.A
        SOP717.MotorREV -> SetIdleSpeed.B
        SOP717.MotorFWD -> SetMotorSafetyBreaker.FWD
        SOP717.MotorREV -> SetMotorSafetyBreaker.REV
        ErrorCheckAndBlockingMotorsAndErrorResetLogic.Output -> SetIdleSpeedToConveyor.Execute
        SOP717.ResetError -> ErrorCheckAndBlockingMotorsAndErrorResetLogic.Reset
        SOP717.MotorFWD -> NoErrorAllowFWD.FWD
        ErrorCheckAndBlockingMotorsAndErrorResetLogic.Output -> NoErrorAllowFWD.Error
        NoErrorAllowFWD.Result -> SetForwardSpeedToConveyor.Execute
        SOP717.MotorREV -> NoErrorAllowREV.REV
        ErrorCheckAndBlockingMotorsAndErrorResetLogic.Output -> NoErrorAllowREV.Error
        NoErrorAllowREV.Result -> SetBackwardSpeedToConveyor.Execute
        SetMotorSafetyBreaker.Result -> ErrorCheckAndBlockingMotorsAndErrorResetLogic.Set
        GraphicsHideLogic.Result -> GraphicsHide.Execute
        SOP717.MotorFWD -> GraphicsHideLogic.FWD
        SOP717.MotorREV -> GraphicsHideLogic.REV
        SOP717.MotorFWD -> MotorFeedbackSignalLogic.A
        SOP717.MotorREV -> MotorFeedbackSignalLogic.A
        ErrorCheckAndBlockingMotorsAndErrorResetLogic.Output -> MotorFeedbackSignalLogic.B
        MotorFeedbackSignalLogic.Result -> SOP717.MotorFeedback
        MotorFeedbackSignalLogic.Result -> GraphicsShow.Execute
        ErrorCheckAndBlockingMotorsAndErrorResetLogic.InvOutput -> SOP717.ConveyorError
        SUB610_B1.SensorSignal -> SOP717.BoxSensor
        ?.Result => ?.Count
        ?.Value => ConveyorSurfaceBehaviour.SurfaceVelocity
        ?.Value => ConveyorSurfaceBehaviour.SurfaceVelocity
        ?.Value => ConveyorSurfaceBehaviour.SurfaceVelocity
        ?.Value => ConveyorSurfaceBehaviour.SurfaceVelocity
        ?.Value => ConveyorSurfaceBehaviour.SurfaceVelocity
        ?.Value => ConveyorSurfaceBehaviour.SurfaceVelocity
        SetIdleSpeedToConveyor.Value => ConveyorSurfaceBehaviour.SurfaceVelocity
        SetForwardSpeedToConveyor.Value => ConveyorSurfaceBehaviour.SurfaceVelocity
        SetBackwardSpeedToConveyor.Value => ConveyorSurfaceBehaviour.SurfaceVelocity
        ?.Result => SetForwardSpeedToConveyor.Max
        ?.A => SetBackwardSpeedToConveyor.Min
        ?.Result => SetBackwardSpeedToConveyor.Max
        ?.A => SetForwardSpeedToConveyor.Min
        GraphicsShow.Object => GraphicsHide.Object
        ?.Object => ?.Object
    - ConveyorSurfaceBehaviour [smart component, from Components\PhysicsControl.rslib] at (-701.82, -354.86, 903.18) mm
        properties: Object=ConveyorSurface; Behavior=1; SurfaceVelocity=8.67025159703114E-14
    - SetIdleSpeedToConveyor [smart component, from Components\Random.rslib] at (-701.82, -354.86, 903.18) mm
        properties: Value=8.67025159703114E-14; Min=0; Max=1E-13
    - SetBackwardSpeedToConveyor [smart component, from Components\Random.rslib] at (-701.82, -354.86, 903.18) mm
        properties: Value=-0.69999999999997; Min=-0.7; Max=-0.6999999999999
    - SetForwardSpeedToConveyor [smart component, from Components\Random.rslib] at (-701.82, -354.86, 903.18) mm
        properties: Value=0.500000000094551; Min=0.5; Max=0.5000000001
    - SetIdleSpeed [smart component, from Components\LogicExpression.rslib] at (-701.82, -354.86, 903.18) mm
        properties: Expression=not A and not B
    - SetMotorSafetyBreaker [smart component, from Components\LogicExpression.rslib] at (-701.82, -354.86, 903.18) mm
        properties: Expression=FWD and REV
    - ErrorCheckAndBlockingMotorsAndErrorResetLogic [smart component, from Components\LogicSRLatch.rslib] at (-701.82, -354.86, 903.18) mm
    - NoErrorAllowFWD [smart component, from Components\LogicExpression.rslib] at (-701.82, -354.86, 903.18) mm
        properties: Expression=FWD and not Error
    - NoErrorAllowREV [smart component, from Components\LogicExpression.rslib] at (-701.82, -354.86, 903.18) mm
        properties: Expression=REV and not Error
    - GraphicsShow [smart component, from Components\Show.rslib] at (-701.82, -354.86, 903.18) mm
        properties: Object=OnOffGfx
    - GraphicsHide [smart component, from Components\Hide.rslib] at (-701.82, -354.86, 903.18) mm
        properties: Object=OnOffGfx
    - GraphicsHideLogic [smart component, from Components\LogicExpression.rslib] at (-701.82, -354.86, 903.18) mm
        properties: Expression=not FWD and not REV
    - GraphicsObjects [graphiccomponentgroup] at (83.9, 149.37, 1003.18) mm, rotated rx 0 ry 0 rz -90 deg
      - OnOffGfx [graphiccomponentgroup] at (514.42, -850.96, -110.92) mm, rotated rx 0 ry 0 rz 90 deg
        - Part_5 [part] at (927.42, 264.29, 0) mm, rotated rx 0 ry 0 rz -90 deg, size 50 x 1493.5 x 100 mm
        - Part_6 [part] at (926.46, -134.61, 0) mm, rotated rx 0 ry 0 rz -90 deg, size 50 x 1492.5 x 100 mm
      - ConveyorSurface [part] at (-0.94, 65.23, -516.89) mm, rotated rx 0 ry 0 rz 180 deg, size 356.8 x 1451.8 x 107.9 mm
    - MotorFeedbackSignalLogic [smart component, from Components\LogicExpression.rslib] at (-701.82, -354.86, 903.18) mm
        properties: Expression=A AND NOT B
    - 1500x450x500 [graphiccomponentgroup] at (162.8, -49.34, 486.29) mm, rotated rx 0 ry 0 rz 180 deg
      - GeneratedPart [part] at (0, 0, 380) mm, size 1500 x 50 x 120 mm
      - GeneratedPart_2 [part] at (0, 400, 380) mm, size 1500 x 50 x 120 mm
      - GeneratedPart_3 [part] at (0, 50, 380) mm, size 50 x 350 x 120 mm
      - GeneratedPart_4 [part] at (1450, 50, 380) mm, size 50 x 350 x 120 mm
      - GeneratedPart_5 [part] at (150, 0, 72) mm
      - GeneratedPart_6 [part] at (150, 0, 72) mm
      - GeneratedPart_7 [part] at (150, 400, 72) mm
      - GeneratedPart_8 [part] at (125, 50, 460) mm, rotated rx -90 ry 0 rz 0 deg, size 80 x 79.7 x 350 mm
      - GeneratedPart_9 [part] at (162.5, -50, 0) mm
      - GeneratedPart_10 [part] at (162.5, -50, 0) mm
      - GeneratedPart_11 [part] at (162.5, 400, 0) mm
      - GeneratedPart_12 [part] at (125, 50, 460) mm, rotated rx -90 ry 0 rz 0 deg, size 80 x 79.7 x 350 mm
      - GeneratedPart_13 [part] at (250, 50, 460) mm, rotated rx -90 ry 0 rz 0 deg, size 80 x 79.7 x 350 mm
      - GeneratedPart_14 [part] at (375, 50, 460) mm, rotated rx -90 ry 0 rz 0 deg, size 80 x 79.7 x 350 mm
      - GeneratedPart_15 [part] at (500, 50, 460) mm, rotated rx -90 ry 0 rz 0 deg, size 80 x 79.7 x 350 mm
      - GeneratedPart_16 [part] at (625, 50, 460) mm, rotated rx -90 ry 0 rz 0 deg, size 80 x 79.7 x 350 mm
      - GeneratedPart_17 [part] at (750, 50, 460) mm, rotated rx -90 ry 0 rz 0 deg, size 80 x 79.7 x 350 mm
      - GeneratedPart_18 [part] at (875, 50, 460) mm, rotated rx -90 ry 0 rz 0 deg, size 80 x 79.7 x 350 mm
      - GeneratedPart_19 [part] at (1000, 50, 460) mm, rotated rx -90 ry 0 rz 0 deg, size 80 x 79.7 x 350 mm
      - GeneratedPart_20 [part] at (1125, 50, 460) mm, rotated rx -90 ry 0 rz 0 deg, size 80 x 79.7 x 350 mm
      - GeneratedPart_21 [part] at (1250, 50, 460) mm, rotated rx -90 ry 0 rz 0 deg, size 80 x 79.7 x 350 mm
      - GeneratedPart_22 [part] at (1375, 50, 460) mm, rotated rx -90 ry 0 rz 0 deg, size 80 x 79.7 x 350 mm
      - GeneratedPart_23 [part] at (200, 25, 12) mm
      - GeneratedPart_24 [part] at (200, 25, 12) mm
      - GeneratedPart_25 [part] at (200, 425, 12) mm
      - GeneratedPart_26 [part] at (1266.54, 400, 0) mm
      - GeneratedPart_27 [part] at (1254.04, 0, 72) mm
      - GeneratedPart_28 [part] at (1304.04, 25, 12) mm
      - GeneratedPart_29 [part] at (1266.54, -50, 0) mm
      - GeneratedPart_30 [part] at (1254.04, 400, 72) mm
      - GeneratedPart_31 [part] at (1304.04, 425, 12) mm
      - Part_3 [part] at (1105.7, 0.66, -486.29) mm, size 100 x 550 x 880 mm
      - Part_2 [part] at (0.3, 0.66, -486.29) mm, size 100 x 550 x 880 mm
    - SUB610_B1 [smart component] at (-13.16, -49.69, 870.13) mm, rotated rx 0 ry 0 rz 180 deg
        signals: DO SensorSignal
        connections:
          SensorRay.SensorOut -> ?.Active
          ?.Output -> SUB610_B1.SensorSignal
          SensorRay.SensorOut -> LogicGate.InputA
          GraphicSwitch_2.Output -> LogicGate_2.InputA
          LogicGate_2.Output -> LogicGate.InputB
          LogicGate.Output -> SUB610_B1.SensorSignal
      - SensorRay [smart component, from Components\LineSensor.rslib] at (24.04, 61.94, 174.13) mm
          properties: Start=[0 0 0]; End=[1.02087466601758E-07 0.23805885165687 4.04628539979468E-07]; Radius=0.01; SensedPart=(none); SensedPoint=[0 0 0]; Length=0.238058851657236; Tag=(none)
        - _sensorPart_ [part], size 20 x 238.1 x 20 mm
      - SensorMountWorking [part] at (0, 0, 0) mm, size 50 x 50 x 200 mm
      - GraphicSwitch_2 [smart component, from Components\GraphicSwitch.rslib] at (50, 0, 0) mm
          properties: PartHigh=SensorMountBroken; PartLow=SensorMountWorking
      - SensorMountBroken [part] at (0, 0, 0) mm, size 50 x 50 x 200 mm
      - LogicGate [smart component, from Components\LogicGate.rslib]
          properties: Operator=AND; Delay=0
      - LogicGate_2 [smart component, from Components\LogicGate.rslib]
          properties: Operator=NOT; Delay=0
  - More_Pallets [smart component]
      signals: DI Create_Pallets, DI sensor723, DI DeletePallet
      connections:
        More_Pallets.Create_Pallets -> Source.Execute
        More_Pallets.Create_Pallets -> Source_2.Execute
        More_Pallets.Create_Pallets -> Source_3.Execute
        More_Pallets.Create_Pallets -> Source_4.Execute
        More_Pallets.Create_Pallets -> Source_5.Execute
        Source.Executed -> Queue_3.Enqueue
        Source_2.Executed -> Queue_3.Enqueue
        Source_3.Executed -> Queue_3.Enqueue
        Source_4.Executed -> Queue_3.Enqueue
        Source_5.Executed -> Queue_3.Enqueue
        More_Pallets.sensor723 -> Queue_4.DeleteAll
        CollisionSensor.SensorOut -> Queue.Enqueue
        CollisionSensor_2.SensorOut -> Queue_2.Enqueue
        CollisionSensor_3.SensorOut -> Queue_3.Enqueue
        CollisionSensor_4.SensorOut -> Queue_4.Enqueue
        CollisionSensor_5.SensorOut -> Queue_5.Enqueue
        More_Pallets.sensor723 -> Queue_2.DeleteAll
        More_Pallets.sensor723 -> Queue_3.DeleteAll
        More_Pallets.sensor723 -> Queue_4.DeleteAll
        More_Pallets.sensor723 -> Queue_5.DeleteAll
        CollisionSensor_10.SensorOut -> Queue_5.Enqueue
        CollisionSensor_9.SensorOut -> Queue_4.Enqueue
        CollisionSensor_6.SensorOut -> Queue.Enqueue
        CollisionSensor_7.SensorOut -> Queue_2.Enqueue
        CollisionSensor_8.SensorOut -> Queue_3.Enqueue
        More_Pallets.Create_Pallets -> Queue_6.Enqueue
        LineSensor_2.SensorOut -> Queue.Enqueue
        LineSensor_7.SensorOut -> Queue_2.Enqueue
        LineSensor_8.SensorOut -> Queue_3.Enqueue
        LineSensor_9.SensorOut -> Queue_4.Enqueue
        Sensor_DeletePallet.SensorOut -> Queue.Enqueue
        Queue_3.Front => Queue_4.Back
        Source.Copy => Queue_3.Back
        Source_2.Copy => Queue_3.Back
        Source_3.Copy => Queue_3.Back
        Source_4.Copy => Queue_3.Back
        Source_5.Copy => Queue_3.Back
        Source.Copy => CollisionSensor.Object1
        Source_2.Copy => CollisionSensor_2.Object1
        Source_3.Copy => CollisionSensor_3.Object1
        Source_4.Copy => CollisionSensor_4.Object1
        Source_5.Copy => CollisionSensor_5.Object1
        CollisionSensor_2.Object1 => Queue_2.Back
        CollisionSensor_3.Object1 => Queue_3.Back
        CollisionSensor_4.Object1 => Queue_4.Back
        CollisionSensor_5.Object1 => Queue_5.Back
        CollisionSensor.Object1 => Queue.Back
        Source_2.Copy => Queue_2.Back
        Source_3.Copy => Queue_3.Back
        Source_4.Copy => Queue_4.Back
        Source_5.Copy => Queue_5.Back
        Source.Copy => CollisionSensor_6.Object1
        Source_2.Copy => CollisionSensor_7.Object1
        Source.Copy => Queue_6.Back
        Source_2.Copy => Queue_6.Back
        Source_3.Copy => Queue_6.Back
        Source_4.Copy => Queue_6.Back
        Source_5.Copy => Queue_6.Back
        Source.Copy => LineSensor_2.SensedPart
        LineSensor_2.SensedPart => Queue.Back
        Source_2.Copy => LineSensor_7.SensedPart
        Source_3.Copy => LineSensor_8.SensedPart
        Source_4.Copy => LineSensor_9.SensedPart
        Sensor_DeletePallet.SensedPart => Queue.Back
    - Source [smart component, from Components\Source.rslib]
        properties: Source=EuroPallet (1); Copy=(none); Parent=(none); Position=[5.727 1.685 0.607]; Orientation=[0 0 0]; Transient=false; PhysicsBehavior=3
    - Source_2 [smart component, from Components\Source.rslib]
        properties: Source=EuroPallet (1); Copy=(none); Parent=(none); Position=[5.727 1.685 0.777]; Orientation=[0 0 0]; Transient=false; PhysicsBehavior=3
    - Source_3 [smart component, from Components\Source.rslib]
        properties: Source=EuroPallet (1); Copy=(none); Parent=(none); Position=[5.727 1.685 0.947]; Orientation=[0 0 0]; Transient=false; PhysicsBehavior=3
    - Source_4 [smart component, from Components\Source.rslib]
        properties: Source=EuroPallet (1); Copy=(none); Parent=(none); Position=[5.727 1.685 1.117]; Orientation=[0 0 0]; Transient=false; PhysicsBehavior=3
    - Source_5 [smart component, from Components\Source.rslib]
        properties: Source=EuroPallet (1); Copy=(none); Parent=(none); Position=[5.727 1.685 1.287]; Orientation=[0 0 0]; Transient=false; PhysicsBehavior=3
    - Queue [smart component, from Components\Queue.rslib]
        properties: Back=(none); Front=(none); Queue={5f7da17f-050c-4867-bb5a-8c884b1ab23c};{3cdbbc78-18f5-434b-b400-26ebd0b10035};{4425d564-100a-4205-9c7c-543e5708241a};{ececd2ae-751b-45d0-b5da-bc69544dd414}; NumberOfObjects=1
    - Sensor_DeletePallet [smart component, from Components\LineSensor.rslib]
        properties: Start=[6.244 5.975 0.665]; End=[6.444 5.975 0.665]; Length=0.2; Radius=0; Tag=(none); SensedPart=(none); SensedPoint=[0 0 0]
      - _sensorPart_ [part], size 200 x 0 x 0 mm
  - SOP720 [smart component] at (6299.14, 1696.77, 617) mm, rotated rx 0 ry 0 rz 90 deg
      properties: ForwardSpeed=0.05; ReverseSpeed=-0.05; ConveyorSpeed=0; SpeedForward=0.7; Constant=1E-09; SpeedBackward=-0.6
      signals: DI MotorFWD, DI MotorREV, DO ConveyorError, DI ResetError, DO MotorFeedback, DI RotateFWD, DI RotateREV, DO RotationFeedback, DO PositionSensorB4, DO PositionSensorB5, DO PositionSensorB6, DO Conveyor_Sensor
      connections:
        SetIdleSpeed.Result -> SetIdleSpeedToConveyor.Execute
        SOP720.MotorFWD -> SetIdleSpeed.A
        SOP720.MotorREV -> SetIdleSpeed.B
        SOP720.MotorFWD -> SetMotorSafetyBreaker.FWD
        SOP720.MotorREV -> SetMotorSafetyBreaker.REV
        ErrorCheckAndBlockingMotorsAndErrorResetLogic.Output -> SetIdleSpeedToConveyor.Execute
        SOP720.ResetError -> ErrorCheckAndBlockingMotorsAndErrorResetLogic.Reset
        SOP720.MotorFWD -> NoErrorAllowFWD.FWD
        ErrorCheckAndBlockingMotorsAndErrorResetLogic.Output -> NoErrorAllowFWD.Error
        NoErrorAllowFWD.Result -> SetForwardSpeedToConveyor.Execute
        SOP720.MotorREV -> NoErrorAllowREV.REV
        ErrorCheckAndBlockingMotorsAndErrorResetLogic.Output -> NoErrorAllowREV.Error
        NoErrorAllowREV.Result -> SetBackwardSpeedToConveyor.Execute
        SetMotorSafetyBreaker.Result -> ErrorCheckAndBlockingMotorsAndErrorResetLogic.Set
        GraphicsHideLogic.Result -> GraphicsHide.Execute
        SOP720.MotorFWD -> GraphicsHideLogic.FWD
        SOP720.MotorREV -> GraphicsHideLogic.REV
        SOP720.MotorFWD -> MotorFeedbackSignalLogic.A
        SOP720.MotorREV -> MotorFeedbackSignalLogic.A
        ErrorCheckAndBlockingMotorsAndErrorResetLogic.Output -> MotorFeedbackSignalLogic.B
        MotorFeedbackSignalLogic.Result -> SOP720.MotorFeedback
        MotorFeedbackSignalLogic.Result -> GraphicsShow.Execute
        SOP720.RotateFWD -> ?.Execute
        SOP720.RotateREV -> ?.Execute
        ?.Executing -> SOP720.RotationFeedback
        ?.Executing -> SOP720.RotationFeedback
        ErrorCheckAndBlockingMotorsAndErrorResetLogic.InvOutput -> SOP720.ConveyorError
        SOP720.RotateFWD -> RotatorFWD.Execute
        SOP720.RotateREV -> ?.Execute
        SOP720.RotateREV -> RotatorREV.Execute
        PlaneSensorB4.SensorOut -> SOP720.PositionSensorB4
        PlaneSensorB6.SensorOut -> SOP720.PositionSensorB6
        PlaneSensorB5.SensorOut -> SOP720.PositionSensorB5
        SOP720.RotateFWD -> SOP720.RotationFeedback
        SOP720.RotateREV -> SOP720.RotationFeedback
        SUB200_B1.SensorSignal -> SOP720.Conveyor_Sensor
        SOP720.RotateFWD -> Rotator_2.Execute
        SOP720.RotateREV -> Rotator.Execute
        SetIdleSpeedToConveyor.Value => ConveyorSurfaceBehaviour.SurfaceVelocity
        SetForwardSpeedToConveyor.Value => ConveyorSurfaceBehaviour.SurfaceVelocity
        SetBackwardSpeedToConveyor.Value => ConveyorSurfaceBehaviour.SurfaceVelocity
        GraphicsShow.Object => GraphicsHide.Object
    - ConveyorSurfaceBehaviour [smart component, from Components\PhysicsControl.rslib] at (-850.96, -505.17, -100) mm
        properties: Object=ConveyorSurface; Behavior=2; SurfaceVelocity=0.500000000025169
    - SetIdleSpeedToConveyor [smart component, from Components\Random.rslib] at (-850.96, -505.17, -100) mm
        properties: Value=1.16161818204523E-14; Min=0; Max=1E-13
    - SetBackwardSpeedToConveyor [smart component, from Components\Random.rslib] at (-850.96, -505.17, -100) mm
        properties: Value=-0.699999999999949; Min=-0.7; Max=-0.6999999999999
    - SetForwardSpeedToConveyor [smart component, from Components\Random.rslib] at (-850.96, -505.17, -100) mm
        properties: Value=0.500000000025169; Min=0.5; Max=0.5000000001
    - SetIdleSpeed [smart component, from Components\LogicExpression.rslib] at (-850.96, -505.17, -100) mm
        properties: Expression=not A and not B
    - SetMotorSafetyBreaker [smart component, from Components\LogicExpression.rslib] at (-850.96, -505.17, -100) mm
        properties: Expression=FWD and REV
    - ErrorCheckAndBlockingMotorsAndErrorResetLogic [smart component, from Components\LogicSRLatch.rslib] at (-850.96, -505.17, -100) mm
    - NoErrorAllowFWD [smart component, from Components\LogicExpression.rslib] at (-850.96, -505.17, -100) mm
        properties: Expression=FWD and not Error
    - NoErrorAllowREV [smart component, from Components\LogicExpression.rslib] at (-850.96, -505.17, -100) mm
        properties: Expression=REV and not Error
    - GraphicsShow [smart component, from Components\Show.rslib] at (-850.96, -505.17, -100) mm
        properties: Object=OnOffGfx
    - GraphicsHide [smart component, from Components\Hide.rslib] at (-850.96, -505.17, -100) mm
        properties: Object=OnOffGfx
    - GraphicsHideLogic [smart component, from Components\LogicExpression.rslib] at (-850.96, -505.17, -100) mm
        properties: Expression=not FWD and not REV
    - GraphicsObjects [graphiccomponentgroup] at (0, 0, -261.68) mm, rotated rx 0 ry 0 rz -89.52 deg
      - OnOffGfx [graphiccomponentgroup] at (515.36, -916.19, 165.2) mm, rotated rx 0 ry 0 rz 90 deg
        - FrameE [part] at (221.83, -88.42, -23.07) mm, size 1370 x 50 x 120 mm
        - FrameB [part] at (221.83, 1063.32, -23.07) mm, size 1370 x 50 x 120 mm
        - FrameC [part] at (1741.48, 853.47, -22.72) mm, rotated rx 0 ry 0 rz 120 deg, size 300 x 50 x 120 mm
        - Frame [part] at (115.23, 829.26, -23.07) mm, rotated rx 0 ry 0 rz 60 deg, size 300 x 50 x 120 mm
        - FrameD [part] at (1741.97, 171.27, 96.95) mm, rotated rx 180 ry 0 rz -120 deg, size 300 x 50 x 120 mm
        - FrameF [part] at (115.25, 195.2, 96.56) mm, rotated rx 180 ry 0 rz -60 deg, size 300 x 50 x 120 mm
      - ConveyorSurface [part] at (506.11, -916.19, 149.32) mm, rotated rx 0 ry 0 rz 90 deg, size 1712.3 x 1089.6 x 114.1 mm
      - 1700x1200x500 [graphiccomponentgroup] at (-645.62, 679.63, -249.56) mm
        - GeneratedPart_49 [part] at (100, -125, 460) mm, rotated rx -90 ry 0 rz -90 deg, size 80 x 80 x 1100 mm
        - GeneratedPart_50 [part] at (100, -250, 460) mm, rotated rx -90 ry 0 rz -90 deg, size 80 x 80 x 1100 mm
        - GeneratedPart_51 [part] at (100, -375, 460) mm, rotated rx -90 ry 0 rz -90 deg, size 80 x 80 x 1100 mm
        - GeneratedPart_52 [part] at (100, -500, 460) mm, rotated rx -90 ry 0 rz -90 deg, size 80 x 80 x 1100 mm
        - GeneratedPart_53 [part] at (100, -625, 460) mm, rotated rx -90 ry 0 rz -90 deg, size 80 x 80 x 1100 mm
        - GeneratedPart_54 [part] at (100, -750, 460) mm, rotated rx -90 ry 0 rz -90 deg, size 80 x 80 x 1100 mm
        - GeneratedPart_55 [part] at (100, -875, 460) mm, rotated rx -90 ry 0 rz -90 deg, size 80 x 80 x 1100 mm
        - GeneratedPart_56 [part] at (100, -1000, 460) mm, rotated rx -90 ry 0 rz -90 deg, size 80 x 80 x 1100 mm
        - GeneratedPart_57 [part] at (100, -1125, 460) mm, rotated rx -90 ry 0 rz -90 deg, size 80 x 80 x 1100 mm
        - GeneratedPart_58 [part] at (100, -1250, 460) mm, rotated rx -90 ry 0 rz -90 deg, size 80 x 80 x 1100 mm
        - RollerE [part] at (403.6, 162.24, 460) mm, rotated rx 90 ry 0 rz 90 deg, size 80 x 78 x 500 mm
        - RollerD [part] at (278.02, 0, 460) mm, rotated rx 90 ry 0 rz 90 deg, size 80 x 80 x 750 mm
        - RollerB [part] at (278.02, -1374.95, 460) mm, rotated rx 90 ry 0 rz 90 deg, size 80 x 80 x 750 mm
        - RollerA [part] at (403.6, -1502.19, 460) mm, rotated rx 90 ry 0 rz 90 deg, size 80 x 78 x 500 mm
        - Frame [part] at (331.73, -1480.59, 380) mm, rotated rx 0 ry 0 rz 150 deg, size 300 x 50 x 120 mm
        - FrameB [part] at (97.67, -1373.99, 380) mm, rotated rx 0 ry 0 rz 90 deg, size 1370 x 50 x 120 mm
        - FrameE [part] at (1249.41, -1373.99, 380) mm, rotated rx 0 ry 0 rz 90 deg, size 1370 x 50 x 120 mm
        - FrameD [part] at (989.72, 146.15, 500.02) mm, rotated rx 180 ry 0 rz -30 deg, size 300 x 50 x 120 mm
        - FrameF [part] at (965.78, -1480.57, 499.63) mm, rotated rx 180 ry 0 rz 30 deg, size 300 x 50 x 120 mm
        - FrameC [part] at (307.52, 145.66, 380.35) mm, rotated rx 0 ry 0 rz -150 deg, size 300 x 50 x 120 mm
      - RotatorPlate [part] at (0, 0, -0.93) mm, rotated rx 0 ry 0 rz 90 deg, size 1600 x 1591.2 x 120 mm
      - Activator [part] at (0, 490.23, 155.75) mm, rotated rx 0 ry 0 rz 90 deg, size 50 x 10 x 20 mm
    - MotorFeedbackSignalLogic [smart component, from Components\LogicExpression.rslib] at (-850.96, -505.17, -100) mm
        properties: Expression=A AND NOT B
    - RotatorFWD [smart component, from Components\Rotator.rslib]
        properties: Object=GraphicsObjects; CenterPoint=[0 0 0]; Axis=[0 0 1]; Speed=-0.174532925199433; Reference=Local; ReferenceObject=(none)
    - RotatorREV [smart component, from Components\Rotator.rslib]
        properties: Object=GraphicsObjects; CenterPoint=[0 0 0]; Axis=[0 0 1]; Speed=0.174532925199433; Reference=Local; ReferenceObject=(none)
    - PlaneSensorB5 [smart component, from Components\PlaneSensor.rslib] at (-4.28, -534.63, -102.3) mm
        properties: Origin=[0 0 0]; Axis1=[0.005 0 0]; Axis2=[0 0.1 0]; SensedPart=(none); Tag=(none)
      - _sensorPart_ [part], size 5 x 100 x 0 mm
    - PlaneSensorB4 [smart component, from Components\PlaneSensor.rslib] at (534.63, 9.69, -102.3) mm, rotated rx 0 ry 0 rz 90 deg
        properties: Origin=[0 0 0]; Axis1=[0.002 0 0]; Axis2=[0 0.1 0]; SensedPart=Activator; Tag=(none)
      - _sensorPart_ [part], size 2 x 100 x 0 mm
    - PlaneSensorB6 [smart component, from Components\PlaneSensor.rslib] at (-13.48, 431.85, -102.3) mm
        properties: Origin=[0 0 0]; Axis1=[0.005 0 0]; Axis2=[0 0.1 0]; SensedPart=(none); Tag=(none)
      - _sensorPart_ [part], size 5 x 100 x 0 mm
    - GFX_legs2 [part] at (410.56, -641.07, -516.89) mm, size 100 x 1300 x 260 mm
    - GFX_legs1 [part] at (-488.8, -641.07, -516.89) mm, size 100 x 1300 x 260 mm
    - SUB200_B1 [smart component] at (537.38, 600.15, -101.56) mm, rotated rx 0 ry 0 rz -179.52 deg
        signals: DO SensorSignal
        connections:
          SensorRay.SensorOut -> ?.Active
          ?.Output -> SUB200_B1.SensorSignal
          SensorRay.SensorOut -> SUB200_B1.SensorSignal
      - SensorRay [smart component, from Components\LineSensor.rslib] at (-25.96, 61.94, 174.13) mm
          properties: Start=[0 0 0]; End=[5.96111039252722E-07 0.938058507471307 1.8696271550378E-07]; Radius=0.01; SensedPart=(none); SensedPoint=[0 0 0]; Length=0.938058507471515; Tag=(none)
        - _sensorPart_ [part], size 20 x 938.1 x 20 mm
      - SensorMount [part] at (-50, 0, 0) mm, size 50 x 50 x 200 mm
    - Rotator [smart component, from Components\Rotator.rslib]
        properties: Object=SUB200_B1; CenterPoint=[0 0 0]; Axis=[0 0 1]; Speed=0.174532925199433; Reference=Object; ReferenceObject=GraphicsObjects
    - Rotator_2 [smart component, from Components\Rotator.rslib]
        properties: Object=SUB200_B1; CenterPoint=[0 0 0]; Axis=[0 0 1]; Speed=-0.174532925199433; Reference=Object; ReferenceObject=GraphicsObjects
  - Part_39 [part] at (5750, 2657.48, 605) mm, size 146.9 x 1169.3 x 58.8 mm
  - Part_42 [part] at (6914, 2657.48, 605) mm, size 208.2 x 1169.5 x 55.1 mm
  - Door [mechanism] at (0, 0, 0) mm; joint values [0] (rad or m)
      links: Frame, Door
  - Door [smart component]
      signals: DI OpenDoor, DO DoorClosed, DO DoorOpened
      connections:
        Door.OpenDoor -> JointMover.Execute
        LogicGate.Output -> JointMover_2.Execute
        Door.OpenDoor -> LogicGate.InputA
        JointMover.Executed -> LogicSRLatch.Set
        LogicSRLatch.Output -> Door.DoorOpened
        LogicGate.Output -> LogicSRLatch.Reset
        JointMover_2.Executed -> LogicSRLatch_2.Set
        Door.OpenDoor -> LogicSRLatch_2.Reset
        LogicSRLatch_2.Output -> Door.DoorClosed
        JointMover_2.Executing -> LogicGate_2.InputB
        LogicGate_2.Output -> Door.DoorOpened
        Door.OpenDoor -> LogicGate_2.InputA
    - JointMover [smart component, from Components\JointMover.rslib]
        properties: Mechanism=Door; Relative=false; Duration=2; J1=-1.5707963267949
    - JointMover_2 [smart component, from Components\JointMover.rslib]
        properties: Mechanism=Door; Relative=false; Duration=2; J1=0
    - LogicGate [smart component, from Components\LogicGate.rslib]
        properties: Operator=NOT; Delay=0
    - LogicSRLatch_2 [smart component, from Components\LogicSRLatch.rslib]
    - LogicGate_2 [smart component, from Components\LogicGate.rslib]
        properties: Operator=OR; Delay=0
Attachment: vacuum is attached to IRB4400_60_196__03 / Link6
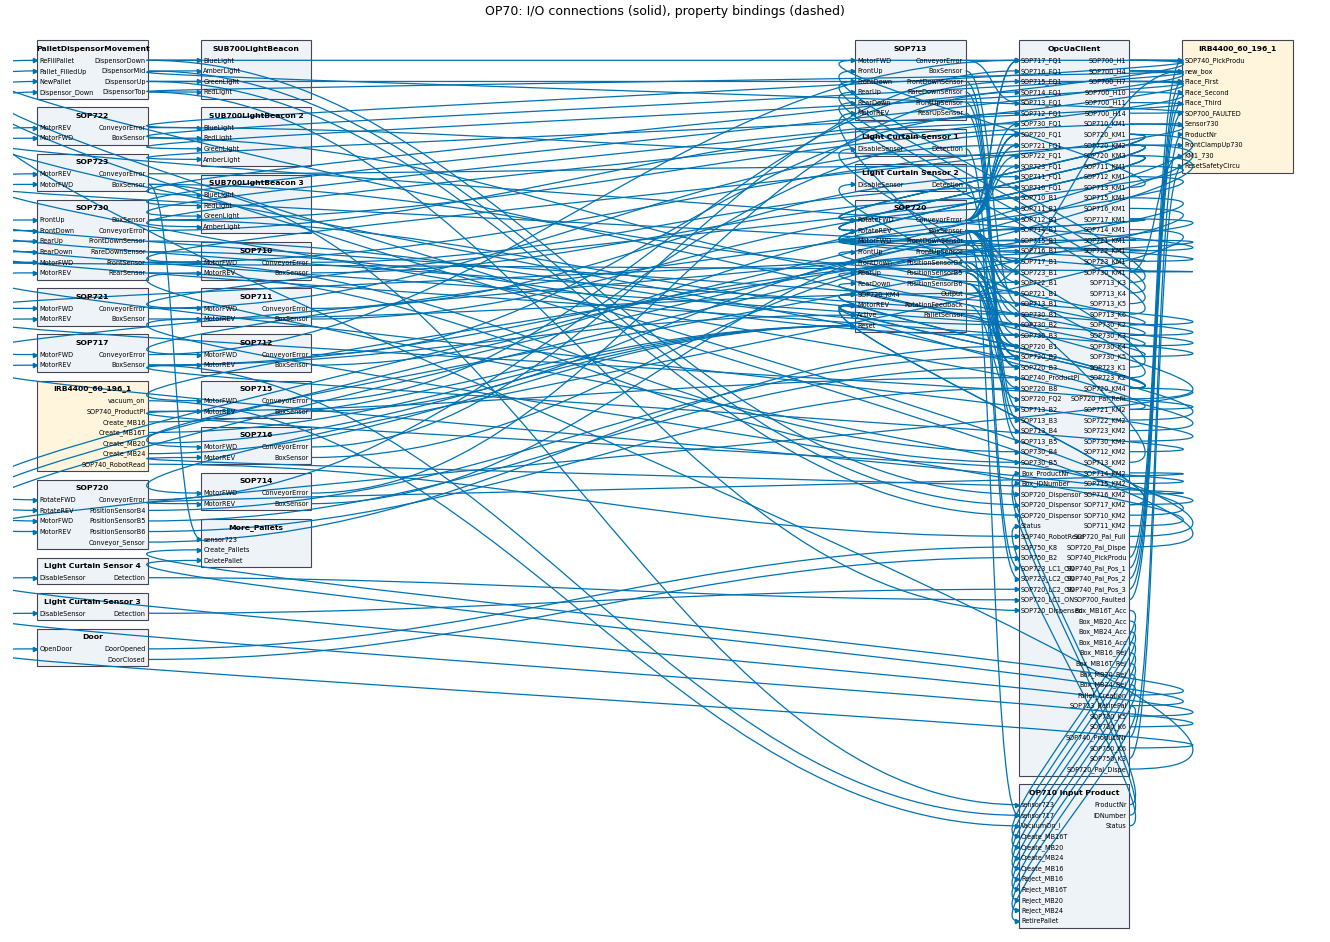
Station logic (signal -> signal, property => property):
  OpcUaClient.SOP700_H1 -> SUB700LightBeacon.BlueLight
  OpcUaClient.SOP700_H1 -> SUB700LightBeacon 2.BlueLight
  OpcUaClient.SOP700_H1 -> SUB700LightBeacon 3.BlueLight
  OpcUaClient.SOP700_H4 -> SUB700LightBeacon 2.RedLight
  OpcUaClient.SOP700_H4 -> SUB700LightBeacon 3.RedLight
  OpcUaClient.SOP700_H7 -> SUB700LightBeacon 2.GreenLight
  OpcUaClient.SOP700_H7 -> SUB700LightBeacon 3.GreenLight
  OpcUaClient.SOP700_H10 -> SUB700LightBeacon 3.AmberLight
  OpcUaClient.SOP700_H11 -> SUB700LightBeacon 2.AmberLight
  OpcUaClient.SOP700_H14 -> SUB700LightBeacon.AmberLight
  OpcUaClient.SOP710_KM1 -> SOP710.MotorFWD
  OpcUaClient.SOP720_KM1 -> SOP720.RotateFWD
  OpcUaClient.SOP720_KM2 -> SOP720.RotateREV
  OpcUaClient.SOP720_KM3 -> SOP720.MotorFWD
  OpcUaClient.SOP711_KM1 -> SOP711.MotorFWD
  OpcUaClient.SOP712_KM1 -> SOP712.MotorFWD
  OpcUaClient.SOP713_KM1 -> SOP713.MotorFWD
  OpcUaClient.SOP715_KM1 -> SOP715.MotorFWD
  OpcUaClient.SOP716_KM1 -> SOP716.MotorFWD
  OpcUaClient.SOP717_KM1 -> SOP717.MotorFWD
  OpcUaClient.SOP714_KM1 -> SOP714.MotorFWD
  SOP717.ConveyorError -> OpcUaClient.SOP717_FQ1
  SOP716.ConveyorError -> OpcUaClient.SOP716_FQ1
  SOP715.ConveyorError -> OpcUaClient.SOP715_FQ1
  SOP714.ConveyorError -> OpcUaClient.SOP714_FQ1
  SOP713.ConveyorError -> OpcUaClient.SOP713_FQ1
  SOP712.ConveyorError -> OpcUaClient.SOP712_FQ1
  SOP730.ConveyorError -> OpcUaClient.SOP730_FQ1
  SOP720.ConveyorError -> OpcUaClient.SOP720_FQ1
  SOP721.ConveyorError -> OpcUaClient.SOP721_FQ1
  SOP722.ConveyorError -> OpcUaClient.SOP722_FQ1
  SOP723.ConveyorError -> OpcUaClient.SOP723_FQ1
  OpcUaClient.SOP721_KM1 -> SOP721.MotorFWD
  OpcUaClient.SOP722_KM1 -> SOP722.MotorFWD
  OpcUaClient.SOP723_KM1 -> SOP723.MotorFWD
  OpcUaClient.SOP730_KM1 -> SOP730.MotorFWD
  SOP711.ConveyorError -> OpcUaClient.SOP711_FQ1
  SOP710.ConveyorError -> OpcUaClient.SOP710_FQ1
